// TIA Portal project "DP_Macko_2024" (V16)

(* hardware
DEVICE "S7-1200 station_1"  S7-1200 Station
   slot 0: "Rack_0"  S7-1200 Rack  Rack  V1.0
   slot 1: "PLC_1"  CPU 1214C DC/DC/DC  6ES7 214-1AG40-0XB0  V4.4
   slot 2: "DQ 16x24VDC_1"  SM 1222 DQ16 x 24VDC  6ES7 222-1BH32-0XB0  V2.0
DEVICE "ET 200SP station_1"  ET 200SP-Station
   slot 0: "Rack_0"  Rack  6ES5 710-8MAx1
   slot 0: "IO device_1"  IM 155-6 PN BA  6ES7 155-6AR00-0AN0  V3.2
   slot 1: "DI 16x24VDC ST_1"  DI 16x24VDC ST  6ES7 131-6BH00-0BA0  V1.1
      slot 1: "DI 16x24VDC ST_1"  DI 16x24VDC ST
   slot 2: "DI 16x24VDC ST_2"  DI 16x24VDC ST  6ES7 131-6BH00-0BA0  V1.1
      slot 1: "DI 16x24VDC ST_2"  DI 16x24VDC ST
   slot 3: "DQ 16x24VDC/0.5A BA_1"  DQ 16x24VDC/0.5A BA  6ES7 132-6BH00-0AA0  V0.0
      slot 1: "DQ 16x24VDC/0.5A BA_1"  DQ 16x24VDC/0.5A BA
   slot 4: "DQ 16x24VDC/0.5A BA_2"  DQ 16x24VDC/0.5A BA  6ES7 132-6BH00-0AA0  V0.0
      slot 1: "DQ 16x24VDC/0.5A BA_2"  DQ 16x24VDC/0.5A BA
   slot 5: "DQ 16x24VDC/0.5A BA_3"  DQ 16x24VDC/0.5A BA  6ES7 132-6BH00-0AA0  V0.0
      slot 1: "DQ 16x24VDC/0.5A BA_3"  DQ 16x24VDC/0.5A BA
   slot 6: "DQ 16x24VDC/0.5A BA_4"  DQ 16x24VDC/0.5A BA  6ES7 132-6BH00-0AA0  V0.0
      slot 1: "DQ 16x24VDC/0.5A BA_4"  DQ 16x24VDC/0.5A BA
   slot 7: "DQ 16x24VDC/0.5A BA_5"  DQ 16x24VDC/0.5A BA  6ES7 132-6BH00-0AA0  V0.0
      slot 1: "DQ 16x24VDC/0.5A BA_5"  DQ 16x24VDC/0.5A BA
   slot 8: "DQ 16x24VDC/0.5A BA_6"  DQ 16x24VDC/0.5A BA  6ES7 132-6BH00-0AA0  V0.0
      slot 1: "DQ 16x24VDC/0.5A BA_6"  DQ 16x24VDC/0.5A BA
   slot 9: "DQ 16x24VDC/0.5A BA_7"  DQ 16x24VDC/0.5A BA  6ES7 132-6BH00-0AA0  V0.0
      slot 1: "DQ 16x24VDC/0.5A BA_7"  DQ 16x24VDC/0.5A BA
   slot 10: "DQ 16x24VDC/0.5A BA_8"  DQ 16x24VDC/0.5A BA  6ES7 132-6BH00-0AA0  V0.0
      slot 1: "DQ 16x24VDC/0.5A BA_8"  DQ 16x24VDC/0.5A BA
   slot 11: "Server module_1"  Server module  6ES7 193-6PA00-0AA0  V1.1
      slot 1: "Server module_1"  Server module
   slot 127: "BA 2xRJ45"  BA 2xRJ45  6ES7 193-6AR00-0AA0  V0.0
      slot 1: "Port_1"  X1 P1 R  6ES7 193-6AR00-0AA0  V0.0
      slot 2: "Port_2"  X1 P2 R  6ES7 193-6AR00-0AA0  V0.0
DEVICE "S7300/ET200M station_1"  S7-300 station
   slot 0: "Rail_0"  Rail  6ES7 390-1***0-0AA0
   slot 2: "PLC_2"  CPU 313C-2 DP  6ES7 313-6CF03-0AB0  V2.6
      slot 0: "MPI interface_1"  X1
      slot 1: "DP interface_1"  X2
      slot 2: "DI 16/DO 16_1"  DI16/DO16
      slot 4: "Count_1"  Counter
   slot 4: "DI 16/DO 16x24VDC/0.5A_1"  DI16/DO16 x 24V / 0.5A  6ES7 323-1BL00-0AA0
   slot 5: "DO 16x24VDC/0.5A_1"  DO16 x 24VDC / 0.5A  6ES7 322-1BH01-0AA0
*)

// ===== PLC "PLC_2"  CPU 313C-2 DP =====

VAR_GLOBAL   // PLC tag table "kolajove_obvody"
   "3k1" AT %I124.4 : Bool;
   "3k2" AT %I124.5 : Bool;
   "4k1" AT %I124.6 : Bool;
   "4k2" AT %I124.7 : Bool;
   "5k1" AT %I125.0 : Bool;
   "5k2" AT %I125.1 : Bool;
   "9k2" AT %I0.1 : Bool;
   "10k1" AT %I0.2 : Bool;
   "10k2" AT %I0.3 : Bool;
   "11k1" AT %I0.4 : Bool;
   "11k2" AT %I0.5 : Bool;
   "8k2" AT %I125.7 : Bool;
   "9k1" AT %I0.0 : Bool;
   "12k1" AT %I0.6 : Bool;
   "12k2" AT %I0.7 : Bool;
   "2k1" AT %I124.2 : Bool;
   "2k2" AT %I124.3 : Bool;
   "6k1" AT %I125.2 : Bool;
   "6k2" AT %I125.3 : Bool;
   "7k1" AT %I125.4 : Bool;
   "14k1" AT %I1.2 : Bool;
   "1k1" AT %I124.0 : Bool;
   "1k2" AT %I124.1 : Bool;
   "7k2" AT %I125.5 : Bool;
   "8k1" AT %I125.6 : Bool;
   "13k1" AT %I1.0 : Bool;
   "13k2" AT %I1.1 : Bool;
   "14k2" AT %I1.3 : Bool;
   "RAD_k1" AT %Q124.0 : Bool;
   "RAD_k2" AT %Q124.1 : Bool;
   "RAD_v1" AT %Q124.2 : Bool;
   "RAD_Sk" AT %Q124.3 : Bool;
   "TU_RAD_ZBE_1" AT %Q124.4 : Bool;
   "TU_RAD_ZBE_2" AT %Q124.5 : Bool;
   "TU_RAD_ZBE_3" AT %Q124.6 : Bool;
   "TU_RAD_ZBE_4" AT %Q124.7 : Bool;
   "ZBE_Lk" AT %Q125.0 : Bool;
   "ZBE_BLk" AT %Q125.1 : Bool;
   "ZBE_v1" AT %Q125.2 : Bool;
   "ZBE_v2" AT %Q125.3 : Bool;
   "ZBE_k1" AT %Q125.4 : Bool;
   "ZBE_k2" AT %Q125.5 : Bool;
   "ZBE_v3" AT %Q125.6 : Bool;
   "ZBE_Sk" AT %Q125.7 : Bool;
   "TU_ZBE_HLO_1" AT %Q0.0 : Bool;
   "TU_ZBE_HLO_2" AT %Q0.1 : Bool;
   "HLO_Lk" AT %Q0.2 : Bool;
   "HLO_v1" AT %Q0.3 : Bool;
   "HLO_k1" AT %Q0.4 : Bool;
   "HLO_k2" AT %Q0.5 : Bool;
   "C_PU1" AT %Q0.7 : Bool;
   "C_AU" AT %Q1.0 : Bool;
   "C_PU2" AT %Q1.1 : Bool;
   "E_PU1" AT %Q1.2 : Bool;
   "E_AU" AT %Q1.3 : Bool;
   "E_PU2" AT %Q1.4 : Bool;
   "OD_ZBE_HLO" AT %Q1.5 : Bool;
END_VAR

DATA_BLOCK "Tratove_useky_DB"   // DB1
{ S7_Optimized_Access := 'FALSE' }
VERSION : 0.1
// stored: InstanceOfName Tratove_useky
"Tratove_useky"
BEGIN
END_DATA_BLOCK

FUNCTION_BLOCK "Tratove_useky"   // FB1, LAD
{ S7_Optimized_Access := 'FALSE' }
VERSION : 0.1
   VAR_INPUT
      RAD_1 : Bool;
      RAD_2 : Bool;
      RAD_3 : Bool;
      RAD_4 : Bool;
      RAD_5 : Bool;
      RAD_ZBE_1 : Bool;
      RAD_ZBE_2 : Bool;
      RAD_ZBE_3 : Bool;
      RAD_ZBE_4 : Bool;
      RAD_ZBE_5 : Bool;
      ZBE_1 : Bool;
      ZBE_2 : Bool;
      ZBE_3 : Bool;
      ZBE_4 : Bool;
      ZBE_5 : Bool;
      ZBE_6 : Bool;
      ZBE_7 : Bool;
      ZBE_8 : Bool;
      ZBE_HLO_1 : Bool;
      ZBE_HLO_2 : Bool;
      ZBE_HLO_3 : Bool;
      ZBE_HLO_4 : Bool;
      ZBE_HLO_5 : Bool;
      ZBE_HLO_6 : Bool;
      HLO_1 : Bool;
      HLO_2 : Bool;
      HLO_3 : Bool;
      HLO_4 : Bool;
   END_VAR
   VAR_OUTPUT
      RAD_k1 : Bool;
      RAD_k2 : Bool;
      RAD_v1 : Bool;
      RAD_Sk : Bool;
      TU_RAD_ZBE_1 : Bool;
      TU_RAD_ZBE_2 : Bool;
      TU_RAD_ZBE_3 : Bool;
      TU_RAD_ZBE_4 : Bool;
      ZBE_Lk : Bool;
      ZBE_BLk : Bool;
      ZBE_v1 : Bool;
      ZBE_v2 : Bool;
      ZBE_k1 : Bool;
      ZBE_k2 : Bool;
      ZBE_v3 : Bool;
      ZBE_Sk : Bool;
      TU_ZBE_HLO_1 : Bool;
      OD_ZBE_HLO : Bool;
      TU_ZBE_HLO_2 : Bool;
      HLO_Lk : Bool;
      HLO_v1 : Bool;
      HLO_k1 : Bool;
      HLO_k2 : Bool;
      C_PU1 : Bool;
      C_AU : Bool;
      C_PU2 : Bool;
      E_PU1 : Bool;
      E_AU : Bool;
      E_PU2 : Bool;
   END_VAR
   VAR
      cRAD_k1 : TON;
      cRAD_k2 : TON;
      cRAD_v1 : TON;
      cRAD_Sk : TON;
      cTU_RAD_ZBE_1 : TON;
      cTU_RAD_ZBE_2 : TON;
      cTU_RAD_ZBE_3 : TON;
      cTU_RAD_ZBE_4 : TON;
      cZBE_Lk : TON;
      cZBE_BLk : TON;
      cZBE_v1 : TON;
      cZBE_v2 : TON;
      cZBE_k1 : TON;
      cZBE_k2 : TON;
      cZBE_v3 : TON;
      cZBE_Sk : TON;
      cTU_ZBE_HLO_1 : TON;
      cOD_ZBE_HLO : TON;
      cTU_ZBE_HLO_2 : TON;
      cHLO_k1 : TON;
      cHLO_k2 : TON;
      cHLO_v1 : TON;
      cHLO_Lk : TON;
      cC_PU1 : TON;
      cC_AU : TON;
      cC_PU2 : TON;
      cE_PU1 : TON;
      cE_AU : TON;
      cE_PU2 : TON;
      oneskorenie : Time := T#250ms;
      cRAD_k1_Off : TON;
      cRAD_k2_Off : TON;
      cRAD_v1_Off : TON;
      cRAD_Sk_Off : TON;
      cTU_RAD_ZBE_1_Off : TON;
      cTU_RAD_ZBE_2_Off : TON;
      cTU_RAD_ZBE_3_Off : TON;
      cTU_RAD_ZBE_4_Off : TON;
      cZBE_Lk_Off : TON;
      cZBE_BLk_Off : TON;
      cZBE_v1_Off : TON;
      cZBE_v2_Off : TON;
      cZBE_k1_Off : TON;
      cZBE_k2_Off : TON;
      cZBE_v3_Off : TON;
      cZBE_Sk_Off : TON;
      cTU_ZBE_HLO_1_Off : TON;
      cOD_ZBE_HLO_Off : TON;
      cTU_ZBE_HLO_2_Off : TON;
      cHLO_k1_Off : TON;
      cHLO_k2_Off : TON;
      cHLO_v1_Off : TON;
      cHLO_Lk_Off : TON;
      cC_PU1_Off : TON;
      cC_AU_Off : TON;
      cC_PU2_Off : TON;
      cE_PU1_Off : TON;
      cE_AU_Off : TON;
      cE_PU2_Off : TON;
   END_VAR
BEGIN

REGION Network 1: Casovac RAD_k1
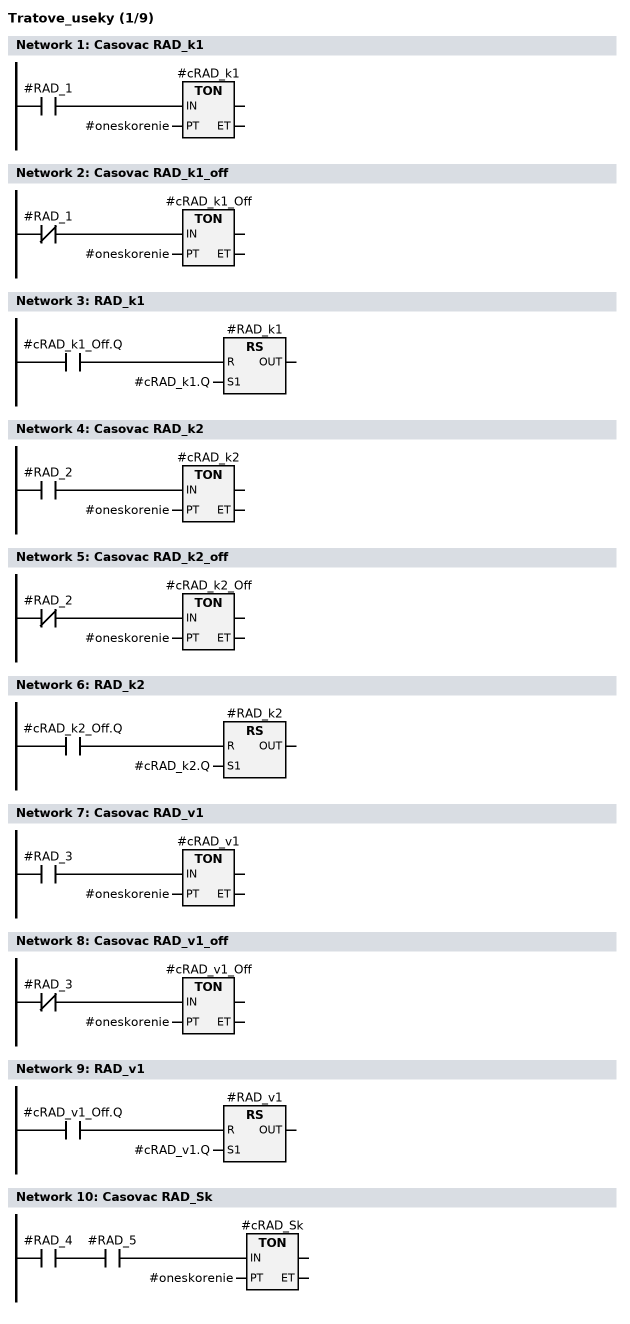
   #cRAD_k1.TON(IN := #RAD_1, PT := #oneskorenie);
END_REGION

REGION Network 2: Casovac RAD_k1_off
   #cRAD_k1_Off.TON(IN := NOT #RAD_1, PT := #oneskorenie);
END_REGION

REGION Network 3: RAD_k1
   RUNG wire#powerrail
      Contact( #cRAD_k1_Off.Q )
      S_RS(operand := #RAD_k1, s1 := #cRAD_k1.Q)
   END_RUNG
   // the same network as SCL:
   IF #cRAD_k1_Off.Q THEN
       #RAD_k1 := FALSE;   // RS flip-flop
   END_IF;
   IF #cRAD_k1.Q THEN #RAD_k1 := TRUE; END_IF;
END_REGION

REGION Network 4: Casovac RAD_k2
   #cRAD_k2.TON(IN := #RAD_2, PT := #oneskorenie);
END_REGION

REGION Network 5: Casovac RAD_k2_off
   #cRAD_k2_Off.TON(IN := NOT #RAD_2, PT := #oneskorenie);
END_REGION

REGION Network 6: RAD_k2
   RUNG wire#powerrail
      Contact( #cRAD_k2_Off.Q )
      S_RS(operand := #RAD_k2, s1 := #cRAD_k2.Q)
   END_RUNG
   // the same network as SCL:
   IF #cRAD_k2_Off.Q THEN
       #RAD_k2 := FALSE;   // RS flip-flop
   END_IF;
   IF #cRAD_k2.Q THEN #RAD_k2 := TRUE; END_IF;
END_REGION

REGION Network 7: Casovac RAD_v1
   #cRAD_v1.TON(IN := #RAD_3, PT := #oneskorenie);
END_REGION

REGION Network 8: Casovac RAD_v1_off
   #cRAD_v1_Off.TON(IN := NOT #RAD_3, PT := #oneskorenie);
END_REGION

REGION Network 9: RAD_v1
   RUNG wire#powerrail
      Contact( #cRAD_v1_Off.Q )
      S_RS(operand := #RAD_v1, s1 := #cRAD_v1.Q)
   END_RUNG
   // the same network as SCL:
   IF #cRAD_v1_Off.Q THEN
       #RAD_v1 := FALSE;   // RS flip-flop
   END_IF;
   IF #cRAD_v1.Q THEN #RAD_v1 := TRUE; END_IF;
END_REGION

REGION Network 10: Casovac RAD_Sk
   #cRAD_Sk.TON(IN := #RAD_4 AND #RAD_5, PT := #oneskorenie);
END_REGION

REGION Network 11: Casovac RAD_Sk_off
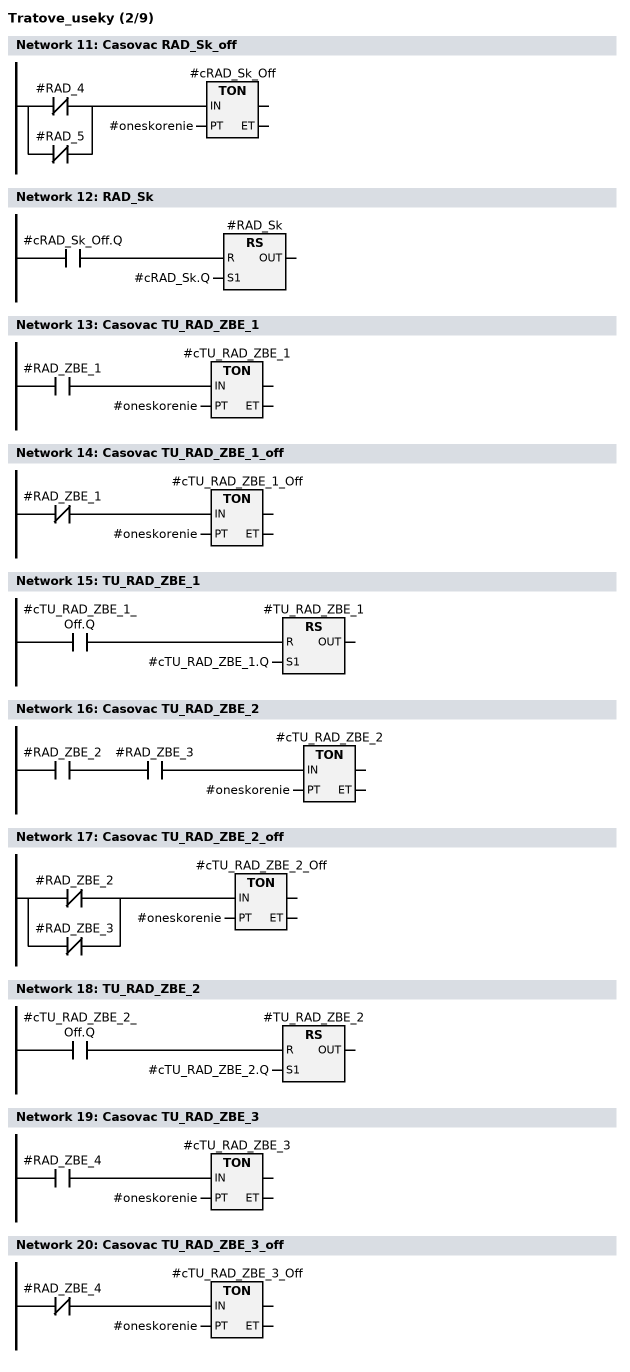
   #cRAD_Sk_Off.TON(IN := NOT #RAD_4 OR NOT #RAD_5, PT := #oneskorenie);
END_REGION

REGION Network 12: RAD_Sk
   RUNG wire#powerrail
      Contact( #cRAD_Sk_Off.Q )
      S_RS(operand := #RAD_Sk, s1 := #cRAD_Sk.Q)
   END_RUNG
   // the same network as SCL:
   IF #cRAD_Sk_Off.Q THEN
       #RAD_Sk := FALSE;   // RS flip-flop
   END_IF;
   IF #cRAD_Sk.Q THEN #RAD_Sk := TRUE; END_IF;
END_REGION

REGION Network 13: Casovac TU_RAD_ZBE_1
   #cTU_RAD_ZBE_1.TON(IN := #RAD_ZBE_1, PT := #oneskorenie);
END_REGION

REGION Network 14: Casovac TU_RAD_ZBE_1_off
   #cTU_RAD_ZBE_1_Off.TON(IN := NOT #RAD_ZBE_1, PT := #oneskorenie);
END_REGION

REGION Network 15: TU_RAD_ZBE_1
   RUNG wire#powerrail
      Contact( #cTU_RAD_ZBE_1_Off.Q )
      S_RS(operand := #TU_RAD_ZBE_1, s1 := #cTU_RAD_ZBE_1.Q)
   END_RUNG
   // the same network as SCL:
   IF #cTU_RAD_ZBE_1_Off.Q THEN
       #TU_RAD_ZBE_1 := FALSE;   // RS flip-flop
   END_IF;
   IF #cTU_RAD_ZBE_1.Q THEN #TU_RAD_ZBE_1 := TRUE; END_IF;
END_REGION

REGION Network 16: Casovac TU_RAD_ZBE_2
   #cTU_RAD_ZBE_2.TON(IN := #RAD_ZBE_2 AND #RAD_ZBE_3, PT := #oneskorenie);
END_REGION

REGION Network 17: Casovac TU_RAD_ZBE_2_off
   #cTU_RAD_ZBE_2_Off.TON(IN := NOT #RAD_ZBE_2 OR NOT #RAD_ZBE_3, PT := #oneskorenie);
END_REGION

REGION Network 18: TU_RAD_ZBE_2
   RUNG wire#powerrail
      Contact( #cTU_RAD_ZBE_2_Off.Q )
      S_RS(operand := #TU_RAD_ZBE_2, s1 := #cTU_RAD_ZBE_2.Q)
   END_RUNG
   // the same network as SCL:
   IF #cTU_RAD_ZBE_2_Off.Q THEN
       #TU_RAD_ZBE_2 := FALSE;   // RS flip-flop
   END_IF;
   IF #cTU_RAD_ZBE_2.Q THEN #TU_RAD_ZBE_2 := TRUE; END_IF;
END_REGION

REGION Network 19: Casovac TU_RAD_ZBE_3
   #cTU_RAD_ZBE_3.TON(IN := #RAD_ZBE_4, PT := #oneskorenie);
END_REGION

REGION Network 20: Casovac TU_RAD_ZBE_3_off
   #cTU_RAD_ZBE_3_Off.TON(IN := NOT #RAD_ZBE_4, PT := #oneskorenie);
END_REGION

REGION Network 21: TU_RAD_ZBE_3
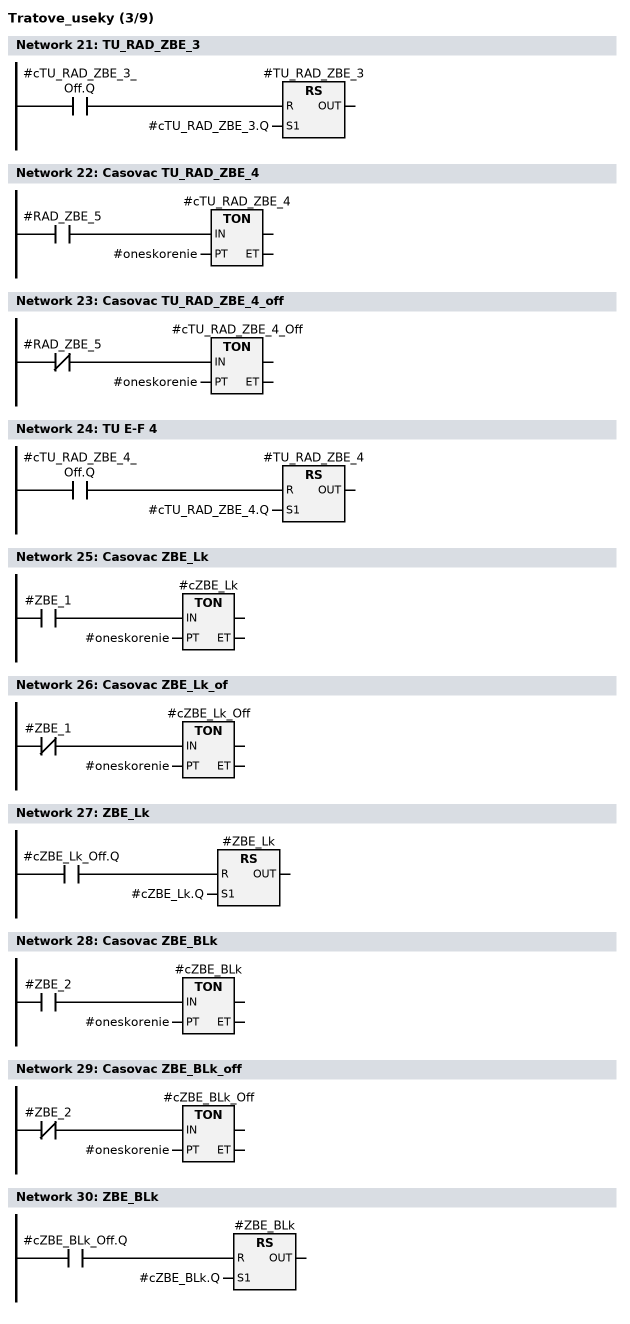
   RUNG wire#powerrail
      Contact( #cTU_RAD_ZBE_3_Off.Q )
      S_RS(operand := #TU_RAD_ZBE_3, s1 := #cTU_RAD_ZBE_3.Q)
   END_RUNG
   // the same network as SCL:
   IF #cTU_RAD_ZBE_3_Off.Q THEN
       #TU_RAD_ZBE_3 := FALSE;   // RS flip-flop
   END_IF;
   IF #cTU_RAD_ZBE_3.Q THEN #TU_RAD_ZBE_3 := TRUE; END_IF;
END_REGION

REGION Network 22: Casovac TU_RAD_ZBE_4
   #cTU_RAD_ZBE_4.TON(IN := #RAD_ZBE_5, PT := #oneskorenie);
END_REGION

REGION Network 23: Casovac TU_RAD_ZBE_4_off
   #cTU_RAD_ZBE_4_Off.TON(IN := NOT #RAD_ZBE_5, PT := #oneskorenie);
END_REGION

REGION Network 24: TU E-F 4
   RUNG wire#powerrail
      Contact( #cTU_RAD_ZBE_4_Off.Q )
      S_RS(operand := #TU_RAD_ZBE_4, s1 := #cTU_RAD_ZBE_4.Q)
   END_RUNG
   // the same network as SCL:
   IF #cTU_RAD_ZBE_4_Off.Q THEN
       #TU_RAD_ZBE_4 := FALSE;   // RS flip-flop
   END_IF;
   IF #cTU_RAD_ZBE_4.Q THEN #TU_RAD_ZBE_4 := TRUE; END_IF;
END_REGION

REGION Network 25: Casovac ZBE_Lk
   #cZBE_Lk.TON(IN := #ZBE_1, PT := #oneskorenie);
END_REGION

REGION Network 26: Casovac ZBE_Lk_of
   #cZBE_Lk_Off.TON(IN := NOT #ZBE_1, PT := #oneskorenie);
END_REGION

REGION Network 27: ZBE_Lk
   RUNG wire#powerrail
      Contact( #cZBE_Lk_Off.Q )
      S_RS(operand := #ZBE_Lk, s1 := #cZBE_Lk.Q)
   END_RUNG
   // the same network as SCL:
   IF #cZBE_Lk_Off.Q THEN
       #ZBE_Lk := FALSE;   // RS flip-flop
   END_IF;
   IF #cZBE_Lk.Q THEN #ZBE_Lk := TRUE; END_IF;
END_REGION

REGION Network 28: Casovac ZBE_BLk
   #cZBE_BLk.TON(IN := #ZBE_2, PT := #oneskorenie);
END_REGION

REGION Network 29: Casovac ZBE_BLk_off
   #cZBE_BLk_Off.TON(IN := NOT #ZBE_2, PT := #oneskorenie);
END_REGION

REGION Network 30: ZBE_BLk
   RUNG wire#powerrail
      Contact( #cZBE_BLk_Off.Q )
      S_RS(operand := #ZBE_BLk, s1 := #cZBE_BLk.Q)
   END_RUNG
   // the same network as SCL:
   IF #cZBE_BLk_Off.Q THEN
       #ZBE_BLk := FALSE;   // RS flip-flop
   END_IF;
   IF #cZBE_BLk.Q THEN #ZBE_BLk := TRUE; END_IF;
END_REGION

REGION Network 31: Casovac ZBE_v1
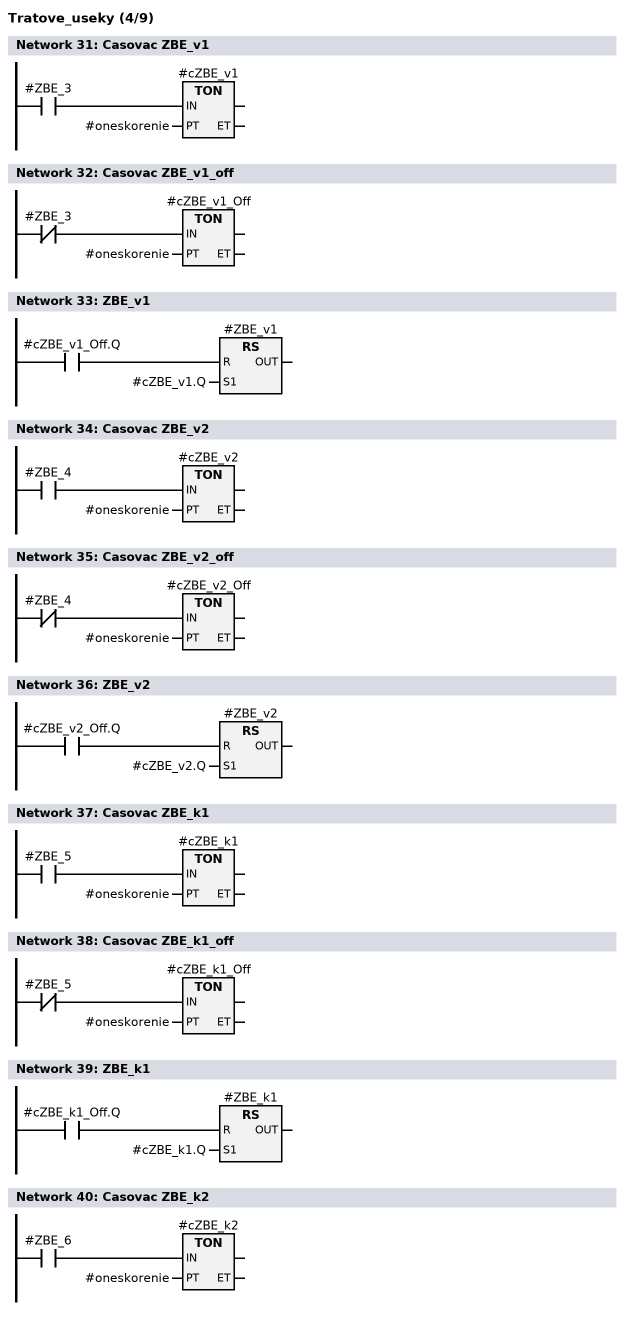
   #cZBE_v1.TON(IN := #ZBE_3, PT := #oneskorenie);
END_REGION

REGION Network 32: Casovac ZBE_v1_off
   #cZBE_v1_Off.TON(IN := NOT #ZBE_3, PT := #oneskorenie);
END_REGION

REGION Network 33: ZBE_v1
   RUNG wire#powerrail
      Contact( #cZBE_v1_Off.Q )
      S_RS(operand := #ZBE_v1, s1 := #cZBE_v1.Q)
   END_RUNG
   // the same network as SCL:
   IF #cZBE_v1_Off.Q THEN
       #ZBE_v1 := FALSE;   // RS flip-flop
   END_IF;
   IF #cZBE_v1.Q THEN #ZBE_v1 := TRUE; END_IF;
END_REGION

REGION Network 34: Casovac ZBE_v2
   #cZBE_v2.TON(IN := #ZBE_4, PT := #oneskorenie);
END_REGION

REGION Network 35: Casovac ZBE_v2_off
   #cZBE_v2_Off.TON(IN := NOT #ZBE_4, PT := #oneskorenie);
END_REGION

REGION Network 36: ZBE_v2
   RUNG wire#powerrail
      Contact( #cZBE_v2_Off.Q )
      S_RS(operand := #ZBE_v2, s1 := #cZBE_v2.Q)
   END_RUNG
   // the same network as SCL:
   IF #cZBE_v2_Off.Q THEN
       #ZBE_v2 := FALSE;   // RS flip-flop
   END_IF;
   IF #cZBE_v2.Q THEN #ZBE_v2 := TRUE; END_IF;
END_REGION

REGION Network 37: Casovac ZBE_k1
   #cZBE_k1.TON(IN := #ZBE_5, PT := #oneskorenie);
END_REGION

REGION Network 38: Casovac ZBE_k1_off
   #cZBE_k1_Off.TON(IN := NOT #ZBE_5, PT := #oneskorenie);
END_REGION

REGION Network 39: ZBE_k1
   RUNG wire#powerrail
      Contact( #cZBE_k1_Off.Q )
      S_RS(operand := #ZBE_k1, s1 := #cZBE_k1.Q)
   END_RUNG
   // the same network as SCL:
   IF #cZBE_k1_Off.Q THEN
       #ZBE_k1 := FALSE;   // RS flip-flop
   END_IF;
   IF #cZBE_k1.Q THEN #ZBE_k1 := TRUE; END_IF;
END_REGION

REGION Network 40: Casovac ZBE_k2
   #cZBE_k2.TON(IN := #ZBE_6, PT := #oneskorenie);
END_REGION

REGION Network 41: Casovac ZBE_k2_off
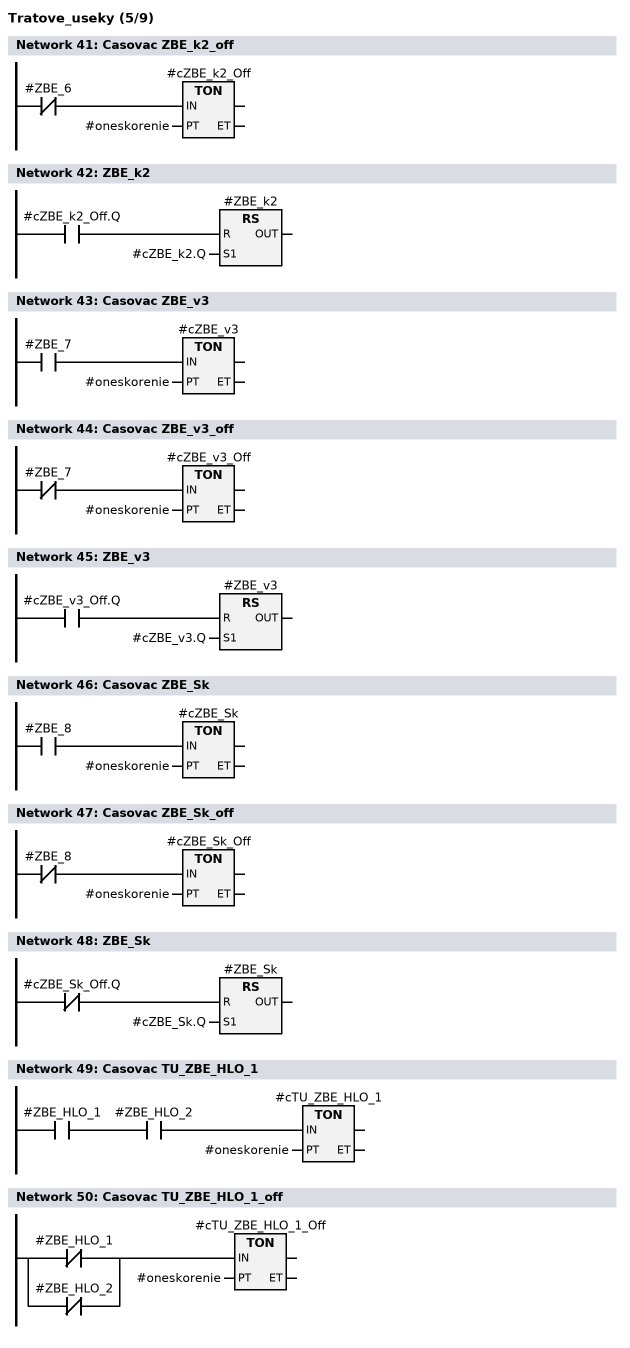
   #cZBE_k2_Off.TON(IN := NOT #ZBE_6, PT := #oneskorenie);
END_REGION

REGION Network 42: ZBE_k2
   RUNG wire#powerrail
      Contact( #cZBE_k2_Off.Q )
      S_RS(operand := #ZBE_k2, s1 := #cZBE_k2.Q)
   END_RUNG
   // the same network as SCL:
   IF #cZBE_k2_Off.Q THEN
       #ZBE_k2 := FALSE;   // RS flip-flop
   END_IF;
   IF #cZBE_k2.Q THEN #ZBE_k2 := TRUE; END_IF;
END_REGION

REGION Network 43: Casovac ZBE_v3
   #cZBE_v3.TON(IN := #ZBE_7, PT := #oneskorenie);
END_REGION

REGION Network 44: Casovac ZBE_v3_off
   #cZBE_v3_Off.TON(IN := NOT #ZBE_7, PT := #oneskorenie);
END_REGION

REGION Network 45: ZBE_v3
   RUNG wire#powerrail
      Contact( #cZBE_v3_Off.Q )
      S_RS(operand := #ZBE_v3, s1 := #cZBE_v3.Q)
   END_RUNG
   // the same network as SCL:
   IF #cZBE_v3_Off.Q THEN
       #ZBE_v3 := FALSE;   // RS flip-flop
   END_IF;
   IF #cZBE_v3.Q THEN #ZBE_v3 := TRUE; END_IF;
END_REGION

REGION Network 46: Casovac ZBE_Sk
   #cZBE_Sk.TON(IN := #ZBE_8, PT := #oneskorenie);
END_REGION

REGION Network 47: Casovac ZBE_Sk_off
   #cZBE_Sk_Off.TON(IN := NOT #ZBE_8, PT := #oneskorenie);
END_REGION

REGION Network 48: ZBE_Sk
   RUNG wire#powerrail
      I_Contact( #cZBE_Sk_Off.Q )
      S_RS(operand := #ZBE_Sk, s1 := #cZBE_Sk.Q)
   END_RUNG
   // the same network as SCL:
   IF NOT #cZBE_Sk_Off.Q THEN
       #ZBE_Sk := FALSE;   // RS flip-flop
   END_IF;
   IF #cZBE_Sk.Q THEN #ZBE_Sk := TRUE; END_IF;
END_REGION

REGION Network 49: Casovac TU_ZBE_HLO_1
   #cTU_ZBE_HLO_1.TON(IN := #ZBE_HLO_1 AND #ZBE_HLO_2, PT := #oneskorenie);
END_REGION

REGION Network 50: Casovac TU_ZBE_HLO_1_off
   #cTU_ZBE_HLO_1_Off.TON(IN := NOT #ZBE_HLO_1 OR NOT #ZBE_HLO_2, PT := #oneskorenie);
END_REGION

REGION Network 51: TU_ZBE_HLO_1
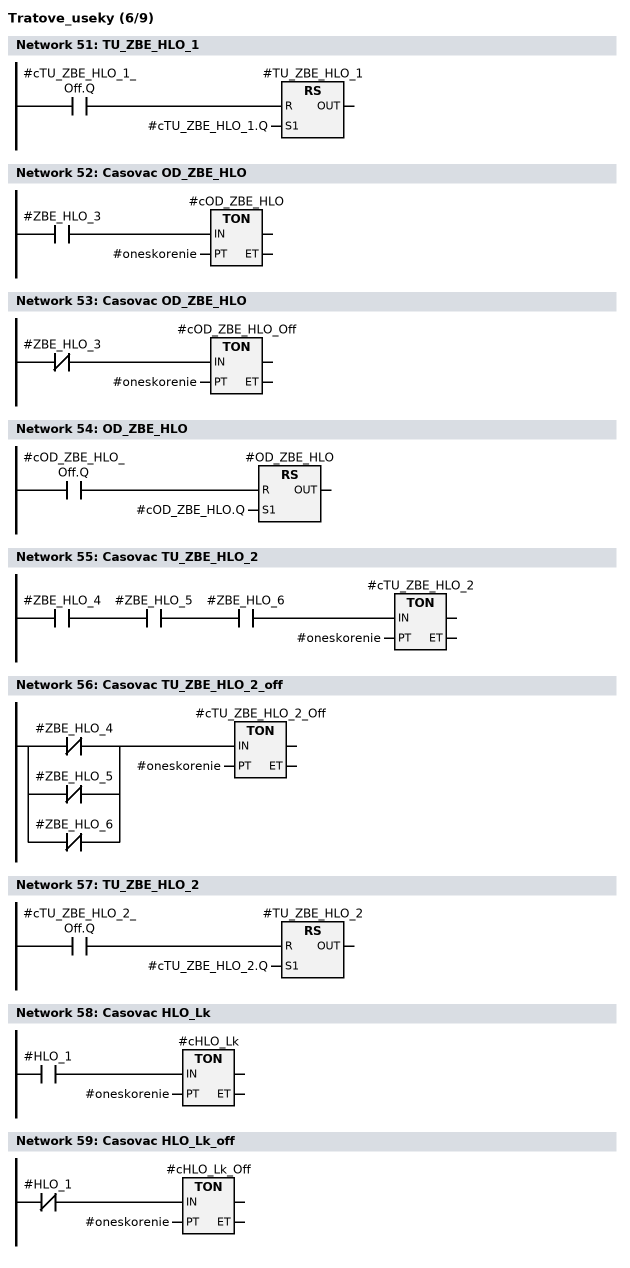
   RUNG wire#powerrail
      Contact( #cTU_ZBE_HLO_1_Off.Q )
      S_RS(operand := #TU_ZBE_HLO_1, s1 := #cTU_ZBE_HLO_1.Q)
   END_RUNG
   // the same network as SCL:
   IF #cTU_ZBE_HLO_1_Off.Q THEN
       #TU_ZBE_HLO_1 := FALSE;   // RS flip-flop
   END_IF;
   IF #cTU_ZBE_HLO_1.Q THEN #TU_ZBE_HLO_1 := TRUE; END_IF;
END_REGION

REGION Network 52: Casovac OD_ZBE_HLO
   #cOD_ZBE_HLO.TON(IN := #ZBE_HLO_3, PT := #oneskorenie);
END_REGION

REGION Network 53: Casovac OD_ZBE_HLO
   #cOD_ZBE_HLO_Off.TON(IN := NOT #ZBE_HLO_3, PT := #oneskorenie);
END_REGION

REGION Network 54: OD_ZBE_HLO
   RUNG wire#powerrail
      Contact( #cOD_ZBE_HLO_Off.Q )
      S_RS(operand := #OD_ZBE_HLO, s1 := #cOD_ZBE_HLO.Q)
   END_RUNG
   // the same network as SCL:
   IF #cOD_ZBE_HLO_Off.Q THEN
       #OD_ZBE_HLO := FALSE;   // RS flip-flop
   END_IF;
   IF #cOD_ZBE_HLO.Q THEN #OD_ZBE_HLO := TRUE; END_IF;
END_REGION

REGION Network 55: Casovac TU_ZBE_HLO_2
   #cTU_ZBE_HLO_2.TON(IN := #ZBE_HLO_4 AND #ZBE_HLO_5 AND #ZBE_HLO_6, PT := #oneskorenie);
END_REGION

REGION Network 56: Casovac TU_ZBE_HLO_2_off
   #cTU_ZBE_HLO_2_Off.TON(IN := NOT #ZBE_HLO_4 OR NOT #ZBE_HLO_5 OR NOT #ZBE_HLO_6, PT := #oneskorenie);
END_REGION

REGION Network 57: TU_ZBE_HLO_2
   RUNG wire#powerrail
      Contact( #cTU_ZBE_HLO_2_Off.Q )
      S_RS(operand := #TU_ZBE_HLO_2, s1 := #cTU_ZBE_HLO_2.Q)
   END_RUNG
   // the same network as SCL:
   IF #cTU_ZBE_HLO_2_Off.Q THEN
       #TU_ZBE_HLO_2 := FALSE;   // RS flip-flop
   END_IF;
   IF #cTU_ZBE_HLO_2.Q THEN #TU_ZBE_HLO_2 := TRUE; END_IF;
END_REGION

REGION Network 58: Casovac HLO_Lk
   #cHLO_Lk.TON(IN := #HLO_1, PT := #oneskorenie);
END_REGION

REGION Network 59: Casovac HLO_Lk_off
   #cHLO_Lk_Off.TON(IN := NOT #HLO_1, PT := #oneskorenie);
END_REGION

REGION Network 60: HLO_Lk
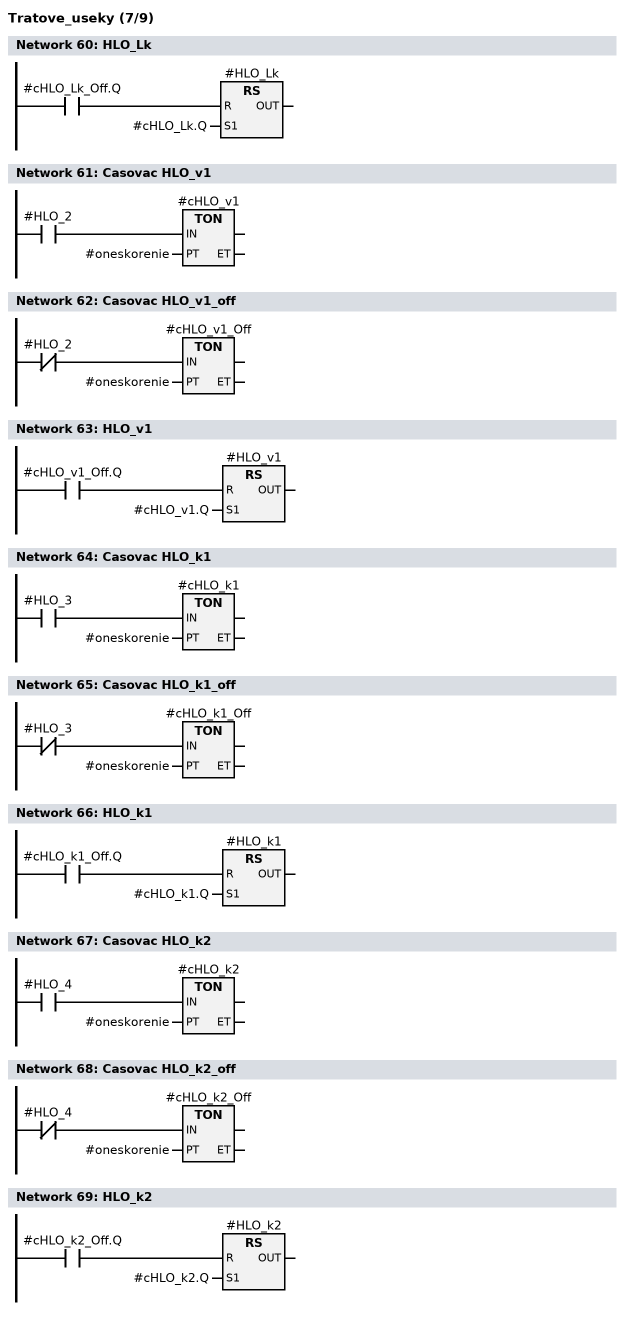
   RUNG wire#powerrail
      Contact( #cHLO_Lk_Off.Q )
      S_RS(operand := #HLO_Lk, s1 := #cHLO_Lk.Q)
   END_RUNG
   // the same network as SCL:
   IF #cHLO_Lk_Off.Q THEN
       #HLO_Lk := FALSE;   // RS flip-flop
   END_IF;
   IF #cHLO_Lk.Q THEN #HLO_Lk := TRUE; END_IF;
END_REGION

REGION Network 61: Casovac HLO_v1
   #cHLO_v1.TON(IN := #HLO_2, PT := #oneskorenie);
END_REGION

REGION Network 62: Casovac HLO_v1_off
   #cHLO_v1_Off.TON(IN := NOT #HLO_2, PT := #oneskorenie);
END_REGION

REGION Network 63: HLO_v1
   RUNG wire#powerrail
      Contact( #cHLO_v1_Off.Q )
      S_RS(operand := #HLO_v1, s1 := #cHLO_v1.Q)
   END_RUNG
   // the same network as SCL:
   IF #cHLO_v1_Off.Q THEN
       #HLO_v1 := FALSE;   // RS flip-flop
   END_IF;
   IF #cHLO_v1.Q THEN #HLO_v1 := TRUE; END_IF;
END_REGION

REGION Network 64: Casovac HLO_k1
   #cHLO_k1.TON(IN := #HLO_3, PT := #oneskorenie);
END_REGION

REGION Network 65: Casovac HLO_k1_off
   #cHLO_k1_Off.TON(IN := NOT #HLO_3, PT := #oneskorenie);
END_REGION

REGION Network 66: HLO_k1
   RUNG wire#powerrail
      Contact( #cHLO_k1_Off.Q )
      S_RS(operand := #HLO_k1, s1 := #cHLO_k1.Q)
   END_RUNG
   // the same network as SCL:
   IF #cHLO_k1_Off.Q THEN
       #HLO_k1 := FALSE;   // RS flip-flop
   END_IF;
   IF #cHLO_k1.Q THEN #HLO_k1 := TRUE; END_IF;
END_REGION

REGION Network 67: Casovac HLO_k2
   #cHLO_k2.TON(IN := #HLO_4, PT := #oneskorenie);
END_REGION

REGION Network 68: Casovac HLO_k2_off
   #cHLO_k2_Off.TON(IN := NOT #HLO_4, PT := #oneskorenie);
END_REGION

REGION Network 69: HLO_k2
   RUNG wire#powerrail
      Contact( #cHLO_k2_Off.Q )
      S_RS(operand := #HLO_k2, s1 := #cHLO_k2.Q)
   END_RUNG
   // the same network as SCL:
   IF #cHLO_k2_Off.Q THEN
       #HLO_k2 := FALSE;   // RS flip-flop
   END_IF;
   IF #cHLO_k2.Q THEN #HLO_k2 := TRUE; END_IF;
END_REGION

REGION Network 70: Casovac C_PU1
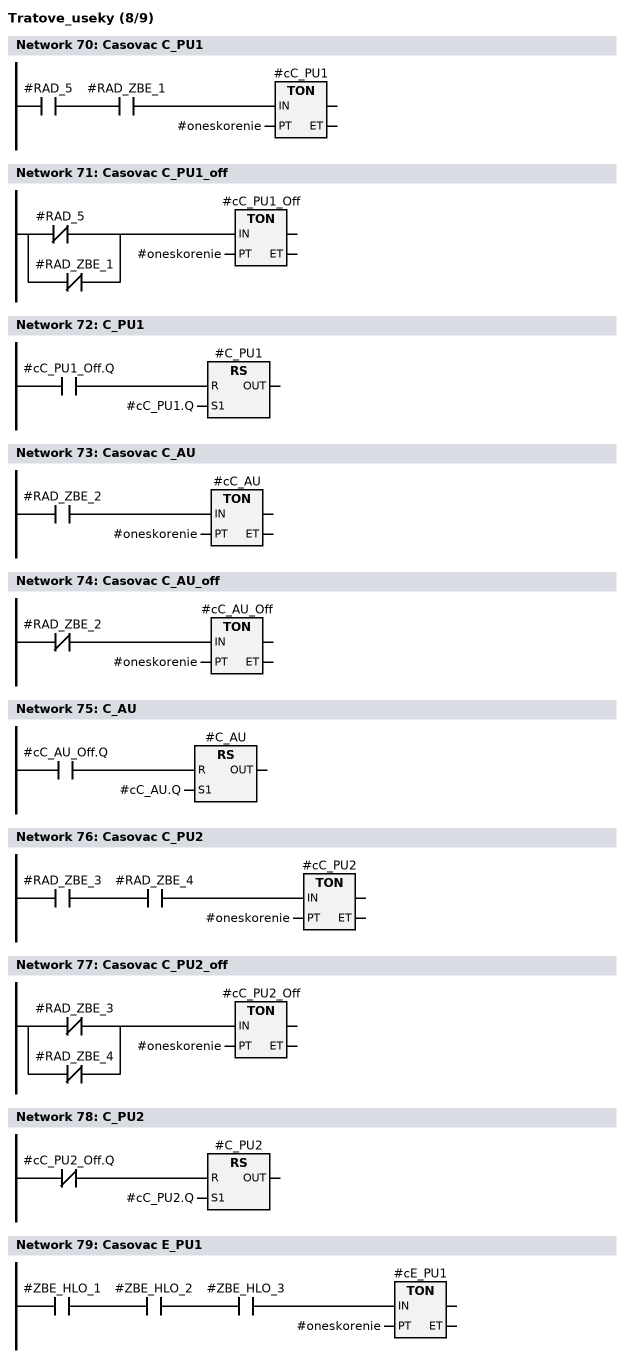
   #cC_PU1.TON(IN := #RAD_5 AND #RAD_ZBE_1, PT := #oneskorenie);
END_REGION

REGION Network 71: Casovac C_PU1_off
   #cC_PU1_Off.TON(IN := NOT #RAD_5 OR NOT #RAD_ZBE_1, PT := #oneskorenie);
END_REGION

REGION Network 72: C_PU1
   RUNG wire#powerrail
      Contact( #cC_PU1_Off.Q )
      S_RS(operand := #C_PU1, s1 := #cC_PU1.Q)
   END_RUNG
   // the same network as SCL:
   IF #cC_PU1_Off.Q THEN
       #C_PU1 := FALSE;   // RS flip-flop
   END_IF;
   IF #cC_PU1.Q THEN #C_PU1 := TRUE; END_IF;
END_REGION

REGION Network 73: Casovac C_AU
   #cC_AU.TON(IN := #RAD_ZBE_2, PT := #oneskorenie);
END_REGION

REGION Network 74: Casovac C_AU_off
   #cC_AU_Off.TON(IN := NOT #RAD_ZBE_2, PT := #oneskorenie);
END_REGION

REGION Network 75: C_AU
   RUNG wire#powerrail
      Contact( #cC_AU_Off.Q )
      S_RS(operand := #C_AU, s1 := #cC_AU.Q)
   END_RUNG
   // the same network as SCL:
   IF #cC_AU_Off.Q THEN
       #C_AU := FALSE;   // RS flip-flop
   END_IF;
   IF #cC_AU.Q THEN #C_AU := TRUE; END_IF;
END_REGION

REGION Network 76: Casovac C_PU2
   #cC_PU2.TON(IN := #RAD_ZBE_3 AND #RAD_ZBE_4, PT := #oneskorenie);
END_REGION

REGION Network 77: Casovac C_PU2_off
   #cC_PU2_Off.TON(IN := NOT #RAD_ZBE_3 OR NOT #RAD_ZBE_4, PT := #oneskorenie);
END_REGION

REGION Network 78: C_PU2
   RUNG wire#powerrail
      I_Contact( #cC_PU2_Off.Q )
      S_RS(operand := #C_PU2, s1 := #cC_PU2.Q)
   END_RUNG
   // the same network as SCL:
   IF NOT #cC_PU2_Off.Q THEN
       #C_PU2 := FALSE;   // RS flip-flop
   END_IF;
   IF #cC_PU2.Q THEN #C_PU2 := TRUE; END_IF;
END_REGION

REGION Network 79: Casovac E_PU1
   #cE_PU1.TON(IN := #ZBE_HLO_1 AND #ZBE_HLO_2 AND #ZBE_HLO_3, PT := #oneskorenie);
END_REGION

REGION Network 80: Casovac E_PU1_off
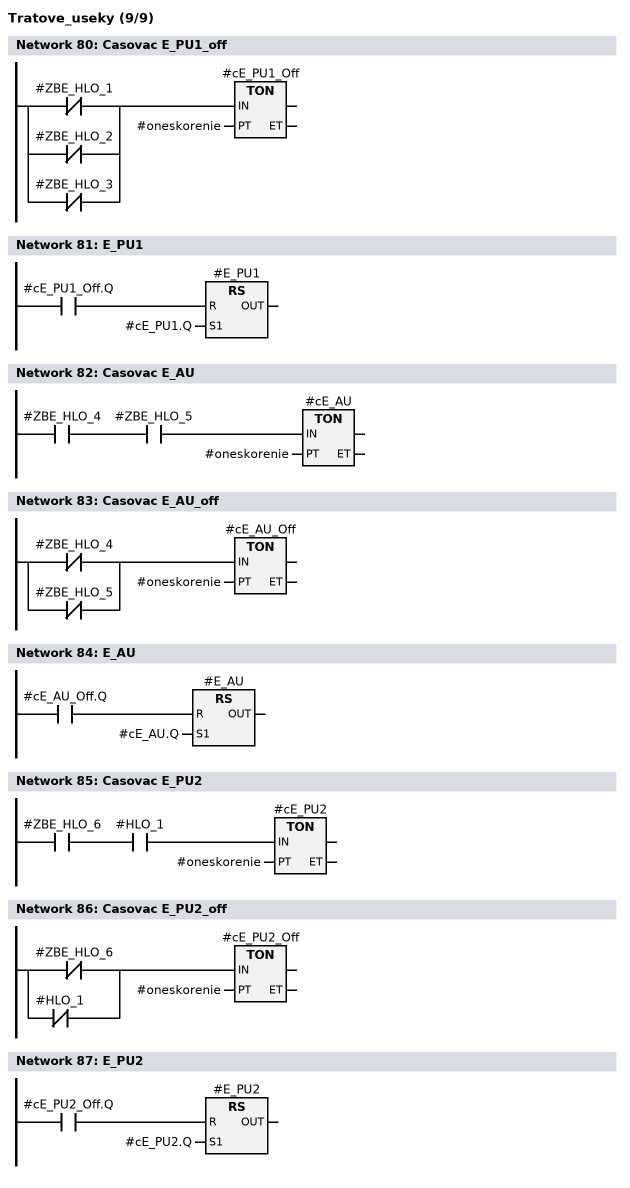
   #cE_PU1_Off.TON(IN := NOT #ZBE_HLO_1 OR NOT #ZBE_HLO_2 OR NOT #ZBE_HLO_3, PT := #oneskorenie);
END_REGION

REGION Network 81: E_PU1
   RUNG wire#powerrail
      Contact( #cE_PU1_Off.Q )
      S_RS(operand := #E_PU1, s1 := #cE_PU1.Q)
   END_RUNG
   // the same network as SCL:
   IF #cE_PU1_Off.Q THEN
       #E_PU1 := FALSE;   // RS flip-flop
   END_IF;
   IF #cE_PU1.Q THEN #E_PU1 := TRUE; END_IF;
END_REGION

REGION Network 82: Casovac E_AU
   #cE_AU.TON(IN := #ZBE_HLO_4 AND #ZBE_HLO_5, PT := #oneskorenie);
END_REGION

REGION Network 83: Casovac E_AU_off
   #cE_AU_Off.TON(IN := NOT #ZBE_HLO_4 OR NOT #ZBE_HLO_5, PT := #oneskorenie);
END_REGION

REGION Network 84: E_AU
   RUNG wire#powerrail
      Contact( #cE_AU_Off.Q )
      S_RS(operand := #E_AU, s1 := #cE_AU.Q)
   END_RUNG
   // the same network as SCL:
   IF #cE_AU_Off.Q THEN
       #E_AU := FALSE;   // RS flip-flop
   END_IF;
   IF #cE_AU.Q THEN #E_AU := TRUE; END_IF;
END_REGION

REGION Network 85: Casovac E_PU2
   #cE_PU2.TON(IN := #ZBE_HLO_6 AND #HLO_1, PT := #oneskorenie);
END_REGION

REGION Network 86: Casovac E_PU2_off
   #cE_PU2_Off.TON(IN := NOT #ZBE_HLO_6 OR NOT #HLO_1, PT := #oneskorenie);
END_REGION

REGION Network 87: E_PU2
   RUNG wire#powerrail
      Contact( #cE_PU2_Off.Q )
      S_RS(operand := #E_PU2, s1 := #cE_PU2.Q)
   END_RUNG
   // the same network as SCL:
   IF #cE_PU2_Off.Q THEN
       #E_PU2 := FALSE;   // RS flip-flop
   END_IF;
   IF #cE_PU2.Q THEN #E_PU2 := TRUE; END_IF;
END_REGION
END_FUNCTION_BLOCK

ORGANIZATION_BLOCK "Main"   // OB1, LAD
TITLE = "Main Program Sweep (Cycle)"
{ S7_Optimized_Access := 'FALSE' }
VERSION : 0.1
   VAR_TEMP
      OB1_EV_CLASS : Byte;   // Bits 0-3 = 1 (Coming event), Bits 4-7 = 1 (Event class 1)
      OB1_SCAN_1 : Byte;   // 1 (Cold restart scan 1 of OB 1), 3 (Scan 2-n of OB 1)
      OB1_PRIORITY : Byte;   // Priority of OB Execution
      OB1_OB_NUMBR : Byte;   // 1 (Organization block 1, OB1)
      OB1_RESERVED_1 : Byte;   // Reserved for system
      OB1_RESERVED_2 : Byte;   // Reserved for system
      OB1_PREV_CYCLE : Int;   // Cycle time of previous OB1 scan (milliseconds)
      OB1_MIN_CYCLE : Int;   // Minimum cycle time of OB1 (milliseconds)
      OB1_MAX_CYCLE : Int;   // Maximum cycle time of OB1 (milliseconds)
      OB1_DATE_TIME : Date_And_Time;   // Date and time OB1 started
   END_VAR
BEGIN

REGION Network 1
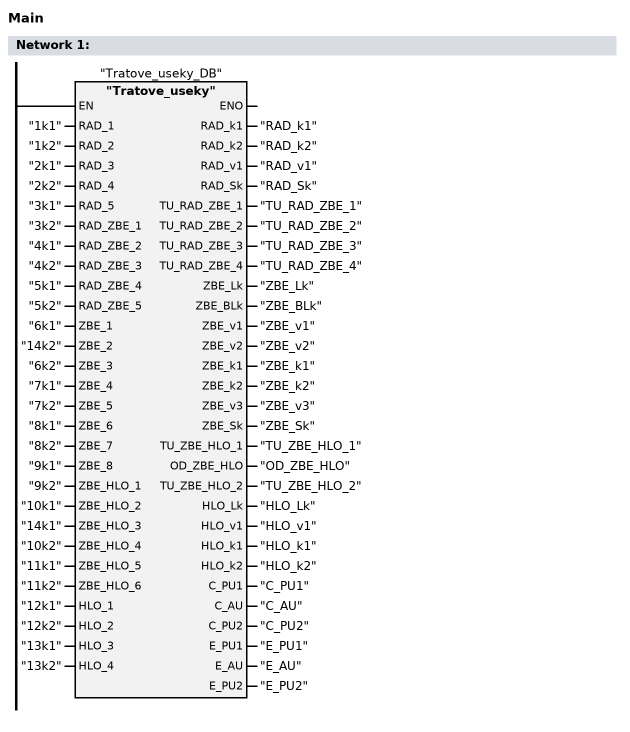
   RUNG wire#powerrail
      "Tratove_useky_DB"(RAD_1 := "1k1", RAD_2 := "1k2", RAD_3 := "2k1", RAD_4 := "2k2", RAD_5 := "3k1", RAD_ZBE_1 := "3k2", RAD_ZBE_2 := "4k1", RAD_ZBE_3 := "4k2", RAD_ZBE_4 := "5k1", RAD_ZBE_5 := "5k2", ZBE_1 := "6k1", ZBE_2 := "14k2", ZBE_3 := "6k2", ZBE_4 := "7k1", ZBE_5 := "7k2", ZBE_6 := "8k1", ZBE_7 := "8k2", ZBE_8 := "9k1", ZBE_HLO_1 := "9k2", ZBE_HLO_2 := "10k1", ZBE_HLO_3 := "14k1", ZBE_HLO_4 := "10k2", ZBE_HLO_5 := "11k1", ZBE_HLO_6 := "11k2", HLO_1 := "12k1", HLO_2 := "12k2", HLO_3 := "13k1", HLO_4 := "13k2", RAD_k1 => "RAD_k1", RAD_k2 => "RAD_k2", RAD_v1 => "RAD_v1", RAD_Sk => "RAD_Sk", TU_RAD_ZBE_1 => "TU_RAD_ZBE_1", TU_RAD_ZBE_2 => "TU_RAD_ZBE_2", TU_RAD_ZBE_3 => "TU_RAD_ZBE_3", TU_RAD_ZBE_4 => "TU_RAD_ZBE_4", ZBE_Lk => "ZBE_Lk", ZBE_BLk => "ZBE_BLk", ZBE_v1 => "ZBE_v1", ZBE_v2 => "ZBE_v2", ZBE_k1 => "ZBE_k1", ZBE_k2 => "ZBE_k2", ZBE_v3 => "ZBE_v3", ZBE_Sk => "ZBE_Sk", TU_ZBE_HLO_1 => "TU_ZBE_HLO_1", OD_ZBE_HLO => "OD_ZBE_HLO", TU_ZBE_HLO_2 => "TU_ZBE_HLO_2", HLO_Lk => "HLO_Lk", HLO_v1 => "HLO_v1", HLO_k1 => "HLO_k1", HLO_k2 => "HLO_k2", C_PU1 => "C_PU1", C_AU => "C_AU", C_PU2 => "C_PU2", E_PU1 => "E_PU1", E_AU => "E_AU", E_PU2 => "E_PU2")
   END_RUNG
   // the same network as SCL:
   "Tratove_useky_DB"(RAD_1 := "1k1",   // "Tratove_useky"
                      RAD_2 := "1k2",
                      RAD_3 := "2k1",
                      RAD_4 := "2k2",
                      RAD_5 := "3k1",
                      RAD_ZBE_1 := "3k2",
                      RAD_ZBE_2 := "4k1",
                      RAD_ZBE_3 := "4k2",
                      RAD_ZBE_4 := "5k1",
                      RAD_ZBE_5 := "5k2",
                      ZBE_1 := "6k1",
                      ZBE_2 := "14k2",
                      ZBE_3 := "6k2",
                      ZBE_4 := "7k1",
                      ZBE_5 := "7k2",
                      ZBE_6 := "8k1",
                      ZBE_7 := "8k2",
                      ZBE_8 := "9k1",
                      ZBE_HLO_1 := "9k2",
                      ZBE_HLO_2 := "10k1",
                      ZBE_HLO_3 := "14k1",
                      ZBE_HLO_4 := "10k2",
                      ZBE_HLO_5 := "11k1",
                      ZBE_HLO_6 := "11k2",
                      HLO_1 := "12k1",
                      HLO_2 := "12k2",
                      HLO_3 := "13k1",
                      HLO_4 := "13k2",
                      RAD_k1 => "RAD_k1",
                      RAD_k2 => "RAD_k2",
                      RAD_v1 => "RAD_v1",
                      RAD_Sk => "RAD_Sk",
                      TU_RAD_ZBE_1 => "TU_RAD_ZBE_1",
                      TU_RAD_ZBE_2 => "TU_RAD_ZBE_2",
                      TU_RAD_ZBE_3 => "TU_RAD_ZBE_3",
                      TU_RAD_ZBE_4 => "TU_RAD_ZBE_4",
                      ZBE_Lk => "ZBE_Lk",
                      ZBE_BLk => "ZBE_BLk",
                      ZBE_v1 => "ZBE_v1",
                      ZBE_v2 => "ZBE_v2",
                      ZBE_k1 => "ZBE_k1",
                      ZBE_k2 => "ZBE_k2",
                      ZBE_v3 => "ZBE_v3",
                      ZBE_Sk => "ZBE_Sk",
                      TU_ZBE_HLO_1 => "TU_ZBE_HLO_1",
                      OD_ZBE_HLO => "OD_ZBE_HLO",
                      TU_ZBE_HLO_2 => "TU_ZBE_HLO_2",
                      HLO_Lk => "HLO_Lk",
                      HLO_v1 => "HLO_v1",
                      HLO_k1 => "HLO_k1",
                      HLO_k2 => "HLO_k2",
                      C_PU1 => "C_PU1",
                      C_AU => "C_AU",
                      C_PU2 => "C_PU2",
                      E_PU1 => "E_PU1",
                      E_AU => "E_AU",
                      E_PU2 => "E_PU2");
END_REGION
END_ORGANIZATION_BLOCK

// ===== PLC "PLC_1"  CPU 1214C DC/DC/DC =====

VAR_GLOBAL   // PLC tag table "Default tag table"
   "Clock_Byte" AT %MB100 : Byte;
   "Clock_10Hz" AT %M100.0 : Bool;
   "Clock_5Hz" AT %M100.1 : Bool;
   "Clock_2.5Hz" AT %M100.2 : Bool;
   "Clock_2Hz" AT %M100.3 : Bool;
   "Clock_1.25Hz" AT %M100.4 : Bool;
   "Clock_1Hz" AT %M100.5 : Bool;
   "Clock_0.625Hz" AT %M100.6 : Bool;
   "Clock_0.5Hz" AT %M100.7 : Bool;
   "TEST" AT %Q16.0 : Bool;
END_VAR

VAR_GLOBAL   // PLC tag table "C_Memory"
   "C_P_PU_BA" AT %M0.5 : Bool;   // Priecestie C: porucha prib useku-smer BA
   "C_P_AU" AT %M0.4 : Bool;   // Priecestie C: porucha anulovacieho useku
   "C_P_PU_AB" AT %M0.3 : Bool;   // Priecestie C: porucha prib. useku-smer AB
   "C_PU_BA" AT %M0.2 : Bool;   // Priecestie C: priblizovaci usek-smer BA
   "C_AU" AT %M0.1 : Bool;   // Priecestie C: anulovaci usek
   "C_PU_AB" AT %M0.0 : Bool;   // Priecestie C: priblizovaci usek-smer AB
   "C_P_Z_H" AT %M0.6 : Bool;   // Priecestie C: porucha zavory hore
   "C_P_Z_D" AT %M0.7 : Bool;   // Priecestie C: porucha zavory dole
   "C_P_C" AT %M1.0 : Bool;   // Priecestie C: porucha cervenej
   "C_P_B" AT %M1.1 : Bool;   // Priecestie C: porucha bielej
   "C_otvorene" AT %M1.2 : Bool;
   "C_zatvorene" AT %M1.3 : Bool;
   "C_predzvananie" AT %M1.4 : Bool;
   "C_manual_zatvor" AT %M3.2 : Bool;
END_VAR

VAR_GLOBAL   // PLC tag table "C_Výstupy"
   "C_C" AT %Q0.0 : Bool;   // Priecestie C: Cervena
   "C_B" AT %Q0.1 : Bool;   // Priecestie C: Biela
   "C_P" AT %Q0.2 : Bool;   // Priecestie C: Porucha
   "C_Z_H" AT %Q0.3 : Bool;   // Priecestie C: Motor Hore
   "C_Z_D" AT %Q0.4 : Bool;   // Priecestie C: Motor Dole
END_VAR

VAR_GLOBAL   // PLC tag table "E_Výstupy"
   "E_C" AT %Q0.5 : Bool;   // Priecestie E: Cervena
   "E_B" AT %Q0.6 : Bool;   // Priecestie E: Biela
   "E_P" AT %Q0.7 : Bool;   // Priecestie E: Porucha
   "E_Z_H" AT %Q1.0 : Bool;   // Priecestie E: Motor Hore
   "E_Z_D" AT %Q1.1 : Bool;   // Priecestie E: Motor Dole
END_VAR

VAR_GLOBAL   // PLC tag table "E_Memory"
   "E_PU_AB" AT %M2.0 : Bool;   // Priecestie E: priblizovaci usek-smer AB
   "E_AU" AT %M2.1 : Bool;   // Priecestie E: anulovaci usek
   "E_PU_BA" AT %M2.2 : Bool;   // Priecestie E: priblizovaciu usek-smer BA
   "E_P_PU_AB" AT %M2.3 : Bool;   // Priecestie E: porucha prib. useku-smer AB
   "E_P_AU" AT %M2.4 : Bool;   // Priecestie E: porucha anulovacieho useku
   "E_P_PU_BA" AT %M2.5 : Bool;   // Priecestie E: porucha prib. useku-smer BA
   "E_P_Z_H" AT %M2.6 : Bool;   // Priecestie E: porucha zavory hore
   "E_P_Z_D" AT %M2.7 : Bool;   // Priecestie E: porucha zavory dole
   "E_P_C" AT %M3.0 : Bool;   // Priecestie E: porucha cervenej
   "E_P_B" AT %M3.1 : Bool;   // Priecestie E: porucha bielej
   "E_otvorene" AT %M1.5 : Bool;
   "E_zatvorene" AT %M1.6 : Bool;
   "E_predzvananie" AT %M1.7 : Bool;
   "E_manual_zatvor" AT %M3.3 : Bool;
END_VAR

VAR_GLOBAL   // PLC tag table "AB-navestidla"
   "AB-18_ze" AT %Q4.0 : Bool;
   "AB-18_ce" AT %Q4.1 : Bool;
   "AB-18_zl" AT %Q3.7 : Bool;
   "AB-19_ze" AT %Q4.3 : Bool;
   "AB-19_ce" AT %Q4.4 : Bool;
   "AB-19_zl" AT %Q4.2 : Bool;
   "AB-28_ze" AT %Q4.6 : Bool;
   "AB-28_ce" AT %Q4.7 : Bool;
   "AB-28_zl" AT %Q4.5 : Bool;
   "AB-29_ze" AT %Q5.1 : Bool;
   "AB-29_ce" AT %Q5.2 : Bool;
   "AB-29_zl" AT %Q5.0 : Bool;
   "AB-39_ze" AT %Q5.4 : Bool;
   "AB-39_ce" AT %Q5.5 : Bool;
   "AB-39_zl" AT %Q5.3 : Bool;
   "AB-40_ze" AT %Q5.7 : Bool;
   "AB-40_ce" AT %Q6.0 : Bool;
   "AB-40_zl" AT %Q5.6 : Bool;
END_VAR

VAR_GLOBAL   // PLC tag table "AH-navestidla"
   "AH-Lo_ze" AT %Q11.6 : Bool;
   "AH-Lo_ce" AT %Q11.7 : Bool;
   "AH-Lo_bi" AT %Q12.0 : Bool;
   "AH-PrLo_ze" AT %Q11.2 : Bool;
   "AH-PrLo_zl" AT %Q11.3 : Bool;
   "AH-So_ze" AT %Q12.1 : Bool;
   "AH-So_ce" AT %Q12.2 : Bool;
   "AH-So_bi" AT %Q12.3 : Bool;
   "AH-PrSo_ze" AT %Q11.4 : Bool;
   "AH-PrSo_zl" AT %Q11.5 : Bool;
END_VAR

VAR_GLOBAL   // PLC tag table "tratove_useky"
   "RAD_k1" AT %I2.0 : Bool;
   "RAD_k2" AT %I2.1 : Bool;
   "RAD_v1" AT %I2.2 : Bool;
   "RAD_Sk" AT %I2.3 : Bool;
   "RAD_ZBE_TU1" AT %I2.4 : Bool;
   "RAD_ZBE_TU2" AT %I2.5 : Bool;
   "RAD_ZBE_TU3" AT %I2.6 : Bool;
   "RAD_ZBE_TU4" AT %I2.7 : Bool;
   "ZBE_Lk" AT %I3.0 : Bool;
   "ZBE_BLk" AT %I3.1 : Bool;
   "ZBE_v1" AT %I3.2 : Bool;
   "ZBE_v2" AT %I3.3 : Bool;
   "ZBE_k1" AT %I3.4 : Bool;
   "ZBE_k2" AT %I3.5 : Bool;
   "ZBE_v3" AT %I3.6 : Bool;
   "ZBE_Sk" AT %I3.7 : Bool;
   "ZBE_HLO_TU1" AT %I4.6 : Bool;
   "ZBE_HLO_TU2" AT %I4.7 : Bool;
   "HLO_Lk" AT %I5.0 : Bool;
   "HLO_v1" AT %I5.1 : Bool;
   "HLO_k1" AT %I5.2 : Bool;
   "HLO_k2" AT %I5.3 : Bool;
   "Priec_C_PU1" AT %I4.0 : Bool;
   "Priec_C_AU" AT %I4.1 : Bool;
   "Priec_C_PU2" AT %I4.2 : Bool;
   "Priec_E_PU1" AT %I4.3 : Bool;
   "Priec_E_AU" AT %I4.4 : Bool;
   "Priec_E_PU2" AT %I4.5 : Bool;
   "ZBE_HLO_OD" AT %I5.4 : Bool;
END_VAR

VAR_GLOBAL   // PLC tag table "St-RAD_navestidla"
   "RAD_L1_zl" AT %Q2.0 : Bool;
   "RAD_L1_ze" AT %Q2.1 : Bool;
   "RAD_L1_ce" AT %Q2.2 : Bool;
   "RAD_L1_bi" AT %Q2.3 : Bool;
   "RAD_L2_zl_h" AT %Q2.4 : Bool;
   "RAD_L2_ze" AT %Q2.5 : Bool;
   "RAD_L2_ce" AT %Q2.6 : Bool;
   "RAD_L2_bi" AT %Q2.7 : Bool;
   "RAD_L2_zl_d" AT %Q3.0 : Bool;
   "RAD_S_zl_h" AT %Q3.3 : Bool;
   "RAD_S_ce" AT %Q3.4 : Bool;
   "RAD_S_bi" AT %Q3.5 : Bool;
   "RAD_S_zl_d" AT %Q3.6 : Bool;
   "RAD_Se1_bi" AT %Q3.1 : Bool;
   "RAD_Se1_mo" AT %Q3.2 : Bool;
   "RAD_stav_L1" AT %MB8 : Byte;
   "RAD_stav_L2" AT %MB9 : Byte;
   "Rad_stav_S" AT %MB10 : Byte;
   "Rad_stav_Se1" AT %MB11 : Byte;
END_VAR

VAR_GLOBAL   // PLC tag table "St-ZBE_navestidla"
   "ZBE_L_zl_h" AT %Q6.1 : Bool;
   "ZBE_L_ze" AT %Q6.2 : Bool;
   "ZBE_L_ce" AT %Q6.3 : Bool;
   "ZBE_L_bi" AT %Q6.4 : Bool;
   "ZBE_L_zl_d" AT %Q6.5 : Bool;
   "ZBE_S1_zl_h" AT %Q7.2 : Bool;
   "ZBE_S1_ze" AT %Q7.3 : Bool;
   "ZBE_S1_ce" AT %Q7.4 : Bool;
   "ZBE_S1_bi" AT %Q7.5 : Bool;
   "ZBE_S2_zl_h" AT %Q7.6 : Bool;
   "ZBE_S2_ze" AT %Q7.7 : Bool;
   "ZBE_S2_ce" AT %Q8.0 : Bool;
   "ZBE_S2_bi" AT %Q8.1 : Bool;
   "ZBE_S2_zl_d" AT %Q8.2 : Bool;
   "ZBE_L1_ze" AT %Q8.3 : Bool;
   "ZBE_L1_ce" AT %Q8.4 : Bool;
   "ZBE_L1_bi" AT %Q8.5 : Bool;
   "ZBE_L2_ze" AT %Q8.6 : Bool;
   "ZBE_L2_ce" AT %Q8.7 : Bool;
   "ZBE_L2_bi" AT %Q9.0 : Bool;
   "ZBE_L2_zl_d" AT %Q9.1 : Bool;
   "ZBE_S_zl_h" AT %Q9.4 : Bool;
   "ZBE_S_ze" AT %Q9.5 : Bool;
   "ZBE_S_ce" AT %Q9.6 : Bool;
   "ZBE_S_bi" AT %Q9.7 : Bool;
   "ZBE_S_zl_d" AT %Q10.0 : Bool;
   "ZBE_Se1_bi" AT %Q6.6 : Bool;
   "ZBE_Se1_mo" AT %Q6.7 : Bool;
   "ZBE_Se2_bi" AT %Q7.0 : Bool;
   "ZBE_Se2_mo" AT %Q7.1 : Bool;
   "ZBE_Se3_bi" AT %Q9.2 : Bool;
   "ZBE_Se3_mo" AT %Q9.3 : Bool;
   "ZBE_PrS_zl" AT %Q10.1 : Bool;
   "ZBE_PrS_ze" AT %Q10.2 : Bool;
   "ZBE_BL_zl_h" AT %Q10.3 : Bool;
   "ZBE_BL_ze" AT %Q10.4 : Bool;
   "ZBE_BL_ce" AT %Q10.5 : Bool;
   "ZBE_BL_bi" AT %Q10.6 : Bool;
   "ZBE_BL_zl_d" AT %Q10.7 : Bool;
   "ZBE_PrBL_zl" AT %Q11.0 : Bool;
   "ZBE_PrBL_ze" AT %Q11.1 : Bool;
   "ZBE_stav_L" AT %MB12 : Byte;
   "ZBE_stav_BL" AT %MB13 : Byte;
   "ZBE_stav_S" AT %MB14 : Byte;
   "ZBE_stav_L1" AT %MB15 : Byte;
   "ZBE_svtav_L2" AT %MB16 : Byte;
   "ZBE_stav_S1" AT %MB17 : Byte;
   "ZBE_stav_S2" AT %MB18 : Byte;
   "ZBE_stav_Se1" AT %MB19 : Byte;
   "ZBE_stav_Se2" AT %MB20 : Byte;
   "ZBE_stav_Se3" AT %MB21 : Byte;
   "ZBE_OD_k1-RAD" AT %M6.0 : Bool;   // Ochranna draha k1 od Radosiny
   "ZBE_OD_k1-HLO" AT %M6.1 : Bool;   // Ochranna draha k1 od Hlohovca
   "ZBE_OD_k2-LUZ" AT %M6.2 : Bool;   // Ochranna draha k2 od Luzianok
   "ZBE_So_navMan" AT %MB28 : Byte;
END_VAR

VAR_GLOBAL   // PLC tag table "St-HLO_navestidla"
   "HLO_PrL_zl" AT %Q12.4 : Bool;
   "HLO_PrL_ze" AT %Q12.5 : Bool;
   "HLO_L_zl_h" AT %Q12.6 : Bool;
   "HLO_L_ce" AT %Q12.7 : Bool;
   "HLO_L_bi" AT %Q13.0 : Bool;
   "HLO_L_zl_d" AT %Q13.1 : Bool;
   "HLO_S1_ze" AT %Q13.4 : Bool;
   "HLO_S1_ce" AT %Q13.5 : Bool;
   "HLO_S1_bi" AT %Q13.6 : Bool;
   "HLO_S2_ze" AT %Q13.7 : Bool;
   "HLO_S2_ce" AT %Q14.0 : Bool;
   "HLO_S2_bi" AT %Q14.1 : Bool;
   "HLO_S2_zl_d" AT %Q14.2 : Bool;
   "HLO_Se1_bi" AT %Q13.3 : Bool;
   "HLO_Se1_mo" AT %Q13.2 : Bool;
   "HLO_stav_L" AT %MB22 : Byte;
   "HLO_stav_S1" AT %MB23 : Byte;
   "HLO_stav_S2" AT %MB24 : Byte;
   "HLO_stav_Se1" AT %MB25 : Byte;
   "HLO_Lo_navMan" AT %MB27 : Byte;
END_VAR

VAR_GLOBAL   // PLC tag table "vyhybky"
   "RAD_vyh1O" AT %Q15.0 : Bool;
   "ZBE_vyh1O" AT %Q15.1 : Bool;
   "ZBE_vyh2O" AT %Q15.2 : Bool;
   "ZBE_vyh3O" AT %Q15.3 : Bool;
   "HLO_vyh1O" AT %Q15.4 : Bool;
   "RAD_vyh1IP" AT %I0.0 : Bool;
   "RAD_vyh1IM" AT %I0.1 : Bool;
   "ZBE_vyh1IP" AT %I0.2 : Bool;
   "ZBE_vyh1IM" AT %I0.3 : Bool;
   "ZBE_vyh2IP" AT %I0.4 : Bool;
   "ZBE_Vyh2IM" AT %I0.5 : Bool;
   "ZBE_vyh3IP" AT %I0.6 : Bool;
   "ZBE_vyh3IM" AT %I0.7 : Bool;
   "HLO_vyh1IP" AT %I1.0 : Bool;
   "HLO_vyh1IM" AT %I1.1 : Bool;
   "ZBE_1-2prestP" AT %M4.2 : Bool;   // Zbe V1-V2: prestavovanie do plusu
   "ZBE_3prestP" AT %M4.4 : Bool;   // Zbe V3: prestavovanie do plusu
   "HLO_1prestP" AT %M4.6 : Bool;   // Hlo V1: prestavovanie do plusu
   "RAD_1prestM" AT %M4.1 : Bool;   // Rad V1: prestavovanie do minusu
   "ZBE_1-2prestM" AT %M4.3 : Bool;   // Zbe V1-V2: prestavovanie do minusu
   "ZBE_3prestM" AT %M4.5 : Bool;   // Zbe V3: prestavovanie do minusu
   "HLO_1prestM" AT %M4.7 : Bool;   // Hlo V1: prestavovanie do minusu
   "RAD_1_smer" AT %M5.0 : Bool;   // Rad V1: smer
   "ZBE_1_smer" AT %M5.4 : Bool;   // Zbe V1: smer
   "ZBE_2_smer" AT %M5.5 : Bool;   // Zbe V2: smer
   "ZBE_3_smer" AT %M5.2 : Bool;   // Zbe V3: smer
   "HLO_1_smer" AT %M5.3 : Bool;   // Hlo V1: smer
   "RAD_1prestP" AT %M4.0 : Bool;   // Rad V1: prestavovanie do plusu
   "ZBE_1-2_smer" AT %M5.1 : Bool;   // Zbe V1-2: smer
   "ZBE_1_prestP" AT %M5.6 : Bool;   // Zbe V1: prestavovanie do plusu
   "ZBE_1_prestM" AT %M5.7 : Bool;   // Zbe V1: prestavovanie do minusu
   "ZBE_2_prestP" AT %M6.3 : Bool;   // Zbe V2: prestavovanie do plusu
   "ZBE_2_prestM" AT %M6.4 : Bool;   // Zbe V2: prestavovanie do minusu
END_VAR

VAR_GLOBAL   // PLC tag table "TS"
   "smer_TS_RAD-ZBE" AT %M7.0 : Bool;   // smer tratoveho suhlasu (0->lichy, 1->sudy)
   "smer_TS_ZBE-HLO" AT %M7.1 : Bool;   // smer tratoveho suhlasu (0->lichy, 1->sudy)
   "volnost_MU_Rad-Zbe" AT %M7.3 : Bool;   // volnost medzist useku RAD - ZBE
   "volnost_MU_Zbe_AH" AT %M7.4 : Bool;   // volnost medzist useku ZBE - AH
   "odchod_RAD" AT %M26.0 : Bool;
   "odchod_ZBE-R" AT %M26.1 : Bool;
   "odchod_ZBE-H" AT %M26.3 : Bool;
   "odchodHLO" AT %M26.4 : Bool;
   "predhlaska_ZBE" AT %M29.0 : Bool;
   "predhlaska_HLO" AT %M29.1 : Bool;
   "odhlaska_ZBE" AT %M29.4 : Bool;
   "odhlaska_HLO" AT %M29.5 : Bool;
   "predhlaska_Lo" AT %M29.2 : Bool;
   "predhlaska_So" AT %M29.3 : Bool;
   "odhlaska_Lo" AT %M29.6 : Bool;
   "odhlaska_So" AT %M29.7 : Bool;
   "volnost_MU_Hlo_AH" AT %M7.5 : Bool;   // volnost medzist useku HLO - AH
END_VAR

DATA_BLOCK "Automaticke_hradlo_Lo"   // DB1
{ S7_Optimized_Access := 'TRUE' }
VERSION : 0.1
// stored: InstanceOfName Automaticke_hradlo
"Automaticke_hradlo"
BEGIN
END_DATA_BLOCK

DATA_BLOCK "Automaticke_hradlo_So"   // DB2
{ S7_Optimized_Access := 'TRUE' }
VERSION : 0.1
// stored: InstanceOfName Automaticke_hradlo
"Automaticke_hradlo"
BEGIN
END_DATA_BLOCK

DATA_BLOCK "Radosina_DB"   // DB3
{ S7_Optimized_Access := 'TRUE' }
VERSION : 0.1
// stored: InstanceOfName Radosina
"Radosina"
BEGIN
END_DATA_BLOCK

DATA_BLOCK "Zbehy_DB"   // DB4
{ S7_Optimized_Access := 'TRUE' }
VERSION : 0.1
// stored: InstanceOfName Zbehy
"Zbehy"
BEGIN
END_DATA_BLOCK

DATA_BLOCK "Hlohovec_DB"   // DB5
{ S7_Optimized_Access := 'TRUE' }
VERSION : 0.1
// stored: InstanceOfName Hlohovec
"Hlohovec"
BEGIN
END_DATA_BLOCK

DATA_BLOCK "Autoblok_18"   // DB6
{ S7_Optimized_Access := 'TRUE' }
VERSION : 0.1
// stored: InstanceOfName Autoblok
"Autoblok"
BEGIN
END_DATA_BLOCK

DATA_BLOCK "Autoblok_19"   // DB7
{ S7_Optimized_Access := 'TRUE' }
VERSION : 0.1
// stored: InstanceOfName Autoblok
"Autoblok"
BEGIN
END_DATA_BLOCK

DATA_BLOCK "Autoblok_28"   // DB8
{ S7_Optimized_Access := 'TRUE' }
VERSION : 0.1
// stored: InstanceOfName Autoblok
"Autoblok"
BEGIN
END_DATA_BLOCK

DATA_BLOCK "Autoblok_29"   // DB9
{ S7_Optimized_Access := 'TRUE' }
VERSION : 0.1
// stored: InstanceOfName Autoblok
"Autoblok"
BEGIN
END_DATA_BLOCK

DATA_BLOCK "Autoblok_40"   // DB10
{ S7_Optimized_Access := 'TRUE' }
VERSION : 0.1
// stored: InstanceOfName Autoblok
"Autoblok"
BEGIN
END_DATA_BLOCK

DATA_BLOCK "Autoblok_39"   // DB11
{ S7_Optimized_Access := 'TRUE' }
VERSION : 0.1
// stored: InstanceOfName Autoblok
"Autoblok"
BEGIN
END_DATA_BLOCK

DATA_BLOCK "Výhybka_RAD1"   // DB12
{ S7_Optimized_Access := 'TRUE' }
VERSION : 0.1
// stored: InstanceOfName Vyhybka
"Vyhybka"
BEGIN
END_DATA_BLOCK

DATA_BLOCK "Výhybka_ZBE1"   // DB13
{ S7_Optimized_Access := 'TRUE' }
VERSION : 0.1
// stored: InstanceOfName Vyhybka
"Vyhybka"
BEGIN
END_DATA_BLOCK

DATA_BLOCK "Výhybka_ZBE2"   // DB14
{ S7_Optimized_Access := 'TRUE' }
VERSION : 0.1
// stored: InstanceOfName Vyhybka
"Vyhybka"
BEGIN
END_DATA_BLOCK

DATA_BLOCK "Výhybka_ZBE3"   // DB15
{ S7_Optimized_Access := 'TRUE' }
VERSION : 0.1
// stored: InstanceOfName Vyhybka
"Vyhybka"
BEGIN
END_DATA_BLOCK

DATA_BLOCK "Výhybka_HLO1"   // DB16
{ S7_Optimized_Access := 'TRUE' }
VERSION : 0.1
// stored: InstanceOfName Vyhybka
"Vyhybka"
BEGIN
END_DATA_BLOCK

DATA_BLOCK "Config"   // DB17
{ S7_Optimized_Access := 'TRUE' }
VERSION : 0.1
   VAR
      Dly_C_PU_AB : Time := T#600ms;   // Oneskorenie v priblizovacom useku AB (C)
      Dly_C_AU : Time := T#600ms;   // Oneskorenie v anulovacom useku (C)
      Dly_C_PU_BA : Time := T#600ms;   // Oneskorenie v priblizovacom useku BA (C)
      AC_C : Time := T#20s;   // Cas anulacie (C)
      VSC_C : Time := T#2500ms;   // Vystrazny sklapaci cas (C)
      ZC_C : Time := T#2500ms;   // Oneskorenie vypnutia svetelnej vysrahy (C)
      Dly_E_PU_AB : Time := T#600ms;   // Oneskorenie v priblizovacom useku AB (E)
      Dly_E_AU : Time := T#600ms;   // Oneskorenie v anulovacom useku (E)
      Dly_E_PU_BA : Time := T#600ms;   // Oneskorenie v priblizovacom useku BA (E)
      AC_E : Time := T#20s;   // Cas anulacie (E)
      VSC_E : Time := T#2500ms;   // Vystrazny sklapaci cas (E)
      ZC_E : Time := T#2500ms;   // Oneskorenie vypnutia svetelnej vystrahy (E)
   END_VAR
BEGIN
END_DATA_BLOCK

DATA_BLOCK "Priecestie_C_DB"   // DB18
{ S7_Optimized_Access := 'TRUE' }
VERSION : 0.1
// stored: InstanceOfName Priecestie
"Priecestie"
BEGIN
END_DATA_BLOCK

DATA_BLOCK "Priecestie_E_DB"   // DB19
{ S7_Optimized_Access := 'TRUE' }
VERSION : 0.1
// stored: InstanceOfName Priecestie
"Priecestie"
BEGIN
END_DATA_BLOCK

FUNCTION_BLOCK "Automaticke_hradlo"   // FB1, LAD
{ S7_Optimized_Access := 'TRUE' }
VERSION : 0.1
   VAR_INPUT
      TS : Bool;
      smerNav : Bool;   // 0-lichy, 1-sudy
      usek_za_nav : Bool;
      usek_pred_nav : Bool;
      navMan : Byte;
      blikac : Bool;
   END_VAR
   VAR_OUTPUT
      zelena : Bool;
      cervena : Bool;
      biela : Bool;
      Pr_zelena : Bool;
      Pr_zlta : Bool;
   END_VAR
   VAR_IN_OUT
      dosla_predhlaska : Bool;
      dosla_odhlaska : Bool;
      odoslana_predhlaska : Bool;
      odoslana_odhlaska : Bool := true;
   END_VAR
   VAR
      stav : Byte;
   END_VAR
   VAR_TEMP   // added for the SCL form of the ladder/FBD networks
      _w1 : Bool;
   END_VAR
BEGIN

REGION Network 1: Zakladny stav
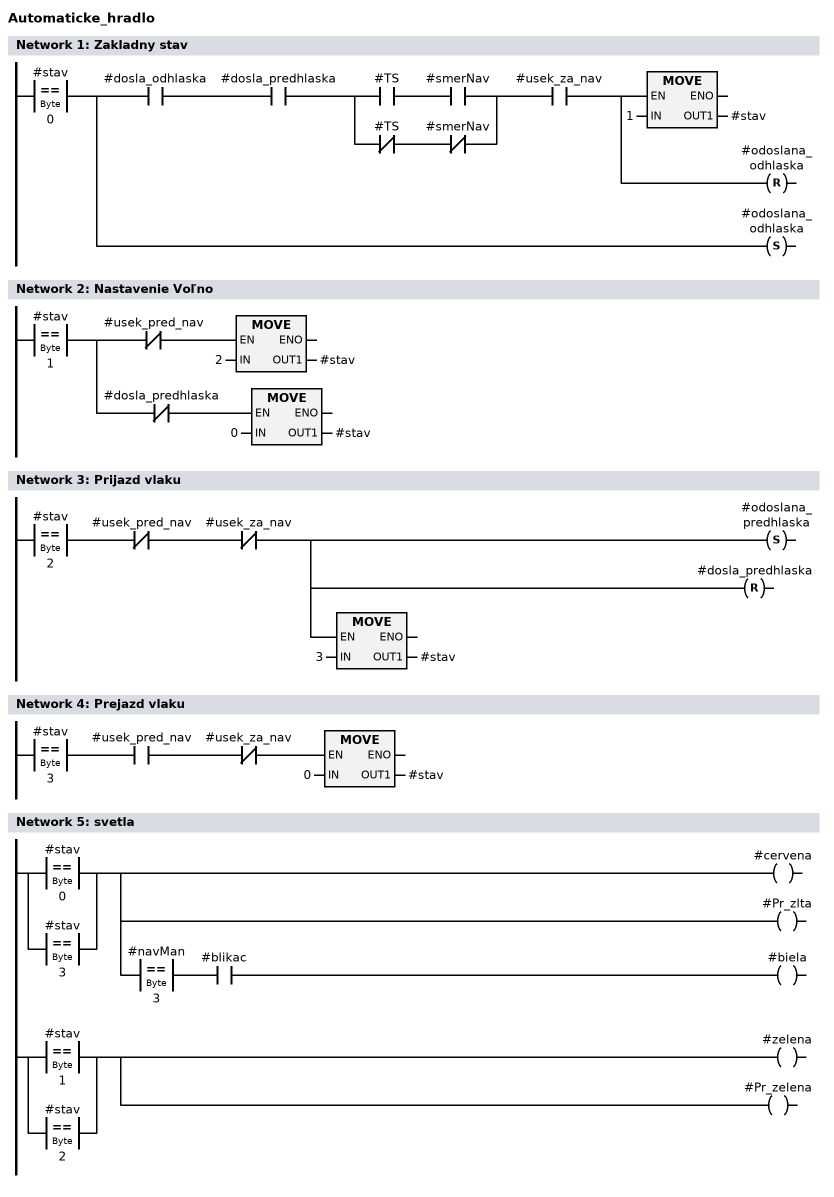
   RUNG wire#powerrail
      { S7_Templates := "SrcType := Byte" } EQ_Contact(in1 := #stav, in2 := 0)
      wire#w1
      Contact( #dosla_odhlaska )
      Contact( #dosla_predhlaska )
      wire#w2
      Contact( #TS )
      Contact( #smerNav )
      wire#w3
      Contact( #usek_za_nav )
      wire#w4
      { S7_GenerateENO := "TRUE" } Move(in := 1, out1 => #stav)
   END_RUNG
   RUNG wire#w2
      I_Contact( #TS )
      I_Contact( #smerNav )
   END_RUNG wire#w3
   RUNG wire#w4
      R_Coil( #odoslana_odhlaska )
   END_RUNG
   RUNG wire#w1
      S_Coil( #odoslana_odhlaska )
   END_RUNG
   // the same network as SCL:
   #_w1 := #stav = 0;
   IF #_w1 AND #dosla_odhlaska AND #dosla_predhlaska AND ((#TS AND #smerNav) OR (NOT #TS AND NOT #smerNav)) AND #usek_za_nav THEN
       #stav := 1;
       #odoslana_odhlaska := FALSE;
   END_IF;
   IF #_w1 THEN #odoslana_odhlaska := TRUE; END_IF;
END_REGION

REGION Network 2: Nastavenie Voľno
   RUNG wire#powerrail
      { S7_Templates := "SrcType := Byte" } EQ_Contact(in1 := #stav, in2 := 1)
      wire#w1
      I_Contact( #usek_pred_nav )
      { S7_GenerateENO := "TRUE" } Move(in := 2, out1 => #stav)
   END_RUNG
   RUNG wire#w1
      I_Contact( #dosla_predhlaska )
      { S7_GenerateENO := "TRUE" } Move(in := 0, out1 => #stav)
   END_RUNG
   // the same network as SCL:
   #_w1 := #stav = 1;
   IF #_w1 AND NOT #usek_pred_nav THEN #stav := 2; END_IF;
   IF #_w1 AND NOT #dosla_predhlaska THEN #stav := 0; END_IF;
END_REGION

REGION Network 3: Prijazd vlaku
   RUNG wire#powerrail
      { S7_Templates := "SrcType := Byte" } EQ_Contact(in1 := #stav, in2 := 2)
      I_Contact( #usek_pred_nav )
      I_Contact( #usek_za_nav )
      wire#w1
      S_Coil( #odoslana_predhlaska )
   END_RUNG
   RUNG wire#w1
      R_Coil( #dosla_predhlaska )
   END_RUNG
   RUNG wire#w1
      { S7_GenerateENO := "TRUE" } Move(in := 3, out1 => #stav)
   END_RUNG
   // the same network as SCL:
   IF (#stav = 2) AND NOT #usek_pred_nav AND NOT #usek_za_nav THEN
       #odoslana_predhlaska := TRUE;
       #dosla_predhlaska := FALSE;
       #stav := 3;
   END_IF;
END_REGION

REGION Network 4: Prejazd vlaku
   RUNG wire#powerrail
      { S7_Templates := "SrcType := Byte" } EQ_Contact(in1 := #stav, in2 := 3)
      Contact( #usek_pred_nav )
      I_Contact( #usek_za_nav )
      { S7_GenerateENO := "TRUE" } Move(in := 0, out1 => #stav)
   END_RUNG
   // the same network as SCL:
   IF (#stav = 3) AND #usek_pred_nav AND NOT #usek_za_nav THEN #stav := 0; END_IF;
END_REGION

REGION Network 5: svetla
   RUNG wire#powerrail
      { S7_Templates := "SrcType := Byte" } EQ_Contact(in1 := #stav, in2 := 0)
      wire#w1
      Coil( #cervena )
   END_RUNG
   RUNG wire#powerrail
      { S7_Templates := "SrcType := Byte" } EQ_Contact(in1 := #stav, in2 := 3)
   END_RUNG wire#w1
   RUNG wire#w1
      Coil( #Pr_zlta )
   END_RUNG
   RUNG wire#w1
      { S7_Templates := "SrcType := Byte" } EQ_Contact(in1 := #navMan, in2 := 3)
      Contact( #blikac )
      Coil( #biela )
   END_RUNG
   RUNG wire#powerrail
      { S7_Templates := "SrcType := Byte" } EQ_Contact(in1 := #stav, in2 := 1)
      wire#w2
      Coil( #zelena )
   END_RUNG
   RUNG wire#powerrail
      { S7_Templates := "SrcType := Byte" } EQ_Contact(in1 := #stav, in2 := 2)
   END_RUNG wire#w2
   RUNG wire#w2
      Coil( #Pr_zelena )
   END_RUNG
   // the same network as SCL:
   #cervena := (#stav = 0) OR (#stav = 3);
   #Pr_zlta := #cervena;
   #biela := #cervena AND (#navMan = 3) AND #blikac;
   #zelena := (#stav = 1) OR (#stav = 2);
   #Pr_zelena := #zelena;
END_REGION
END_FUNCTION_BLOCK

FUNCTION_BLOCK "Priecestie"   // FB2, LAD
{ S7_Optimized_Access := 'TRUE' }
VERSION : 0.1
   VAR_INPUT
      PU_AB : Bool;   // Priblizovaci usek-smer AB
      AU : Bool;   // Anulovaci usek
      PU_BA : Bool;   // Priblizovaci usek-smer BA
      P_Z_H : Bool;   // Porucha zavora hore
      P_Z_D : Bool;   // Porucha zavora dole
      AC : Time;   // Anulovaci cas
      VSC : Time;   // Vystrazny sklapaci cas
      ZC : Time;
      manual : Bool;
   END_VAR
   VAR_OUTPUT
      Z_H : Bool;   // Zavora hore
      Z_D : Bool;   // Zavora dole
      C : Bool;   // Cervena
      "B" : Bool;   // Biela
      predzvananie : Bool;
      priecestie_zatvorene : Bool;
      priecestie_otvorene : Bool;
   END_VAR
   VAR
      S_AB : Bool;   // Smer A->B
      S_BA : Bool;   // Smer B->A
      Vystraha : Bool;   // Spustenie vystrahy
      R_AB : Bool;   // Ukoncenie vystrahy pre smer A->B
      R_BA : Bool;   // Ukoncenie vystrahy pre smer B->A
      R_BBA : Bool;   // Reset vystrahy bez prejazdu priecestia smerom BA
      R_BAB : Bool;   // Reset vystrahy bez prejazdu priecestia smerom AB
      P1 : Bool;   // Pomocna premenna pre otvorenie zavor
      P2 : Bool;   // Pomocna premenna
      P3 : Bool;   // Pomocna premenna
      CA_time : Time;   // Cas anulacie
      CA : TON_TIME;   // Zaznamenanie casu anulacie
      SmerDB : "Detekcia_Smeru_Jazdy";   // Detekcia smeru jazdy KV
      TON1 : TON_TIME;   // Vystrazny sklapaci cas
      TOF1 : TOF_TIME;   // Oneskorenie vypnutia vystrahy vystraznika po anulacii vystrahy
      ZH_ZD : TON_TIME;   // Oneskorenie medzi zdvihanim a spustanim zavor
   END_VAR
   VAR CONSTANT
      ZH_ZD_delay : Time := T#250ms;   // Cas pre oneskorenie medzi zdvihanim a spustanim zavor
   END_VAR
   VAR_TEMP   // added for the SCL form of the ladder/FBD networks
      _w1 : Bool;
      _w2 : Bool;
   END_VAR
BEGIN

REGION Network 1: Vyhodnotenie smeru jazdy KV
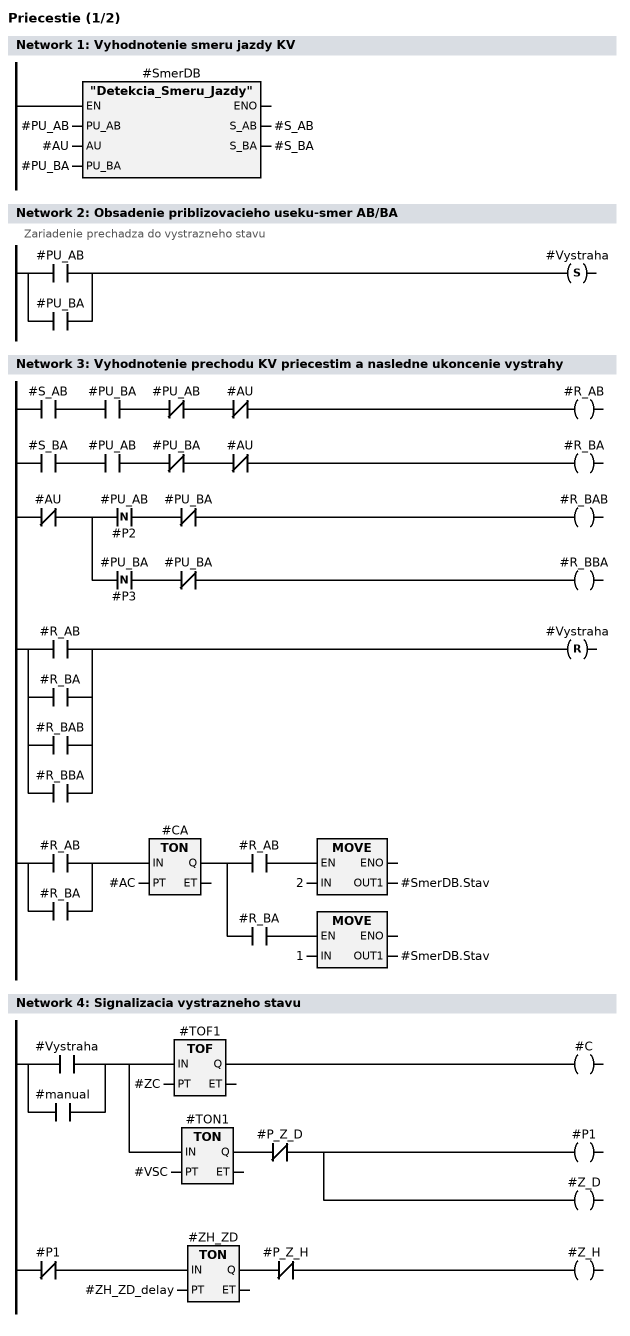
   RUNG wire#powerrail
      #SmerDB(PU_AB := #PU_AB, AU := #AU, PU_BA := #PU_BA, S_AB => #S_AB, S_BA => #S_BA)
   END_RUNG
   // the same network as SCL:
   #SmerDB(PU_AB := #PU_AB, AU := #AU, PU_BA := #PU_BA, S_AB => #S_AB, S_BA => #S_BA);   // "Detekcia_Smeru_Jazdy"
END_REGION

REGION Network 2: Obsadenie priblizovacieho useku-smer AB/BA
   // Zariadenie prechadza do vystrazneho stavu
   RUNG wire#powerrail
      Contact( #PU_AB )
      wire#w1
      S_Coil( #Vystraha )
   END_RUNG
   RUNG wire#powerrail
      Contact( #PU_BA )
   END_RUNG wire#w1
   // the same network as SCL:
   IF #PU_AB OR #PU_BA THEN #Vystraha := TRUE; END_IF;
END_REGION

REGION Network 3: Vyhodnotenie prechodu KV priecestim a nasledne ukoncenie vystrahy
   #R_AB := #S_AB AND #PU_BA AND NOT #PU_AB AND NOT #AU;
   #R_BA := #S_BA AND #PU_AB AND NOT #PU_BA AND NOT #AU;
   #_w1 := NOT #AU AND NOT #PU_AB AND #P2;   // falling edge of #PU_AB
   #P2 := #PU_AB;
   #R_BAB := #_w1 AND NOT #PU_BA;
   #_w2 := NOT #AU AND NOT #PU_BA AND #P3;   // falling edge of #PU_BA
   #P3 := #PU_BA;
   #R_BBA := #_w2 AND NOT #PU_BA;
   IF #R_AB OR #R_BA OR #R_BAB OR #R_BBA THEN #Vystraha := FALSE; END_IF;
   #CA(IN := #R_AB OR #R_BA, PT := #AC);   // TON
   IF #CA.Q AND #R_AB THEN #SmerDB.Stav := 2; END_IF;
   IF #CA.Q AND #R_BA THEN #SmerDB.Stav := 1; END_IF;
END_REGION

REGION Network 4: Signalizacia vystrazneho stavu
   #_w1 := #Vystraha OR #manual;
   #TOF1(IN := #_w1, PT := #ZC);   // TOF
   #C := #TOF1.Q;
   #TON1(IN := #_w1, PT := #VSC);   // TON
   #P1 := #TON1.Q AND NOT #P_Z_D;
   #Z_D := #P1;
   #ZH_ZD(IN := NOT #P1, PT := #ZH_ZD_delay);   // TON
   #Z_H := #ZH_ZD.Q AND NOT #P_Z_H;
END_REGION

REGION Network 5: Signalizacia zakladneho stavu
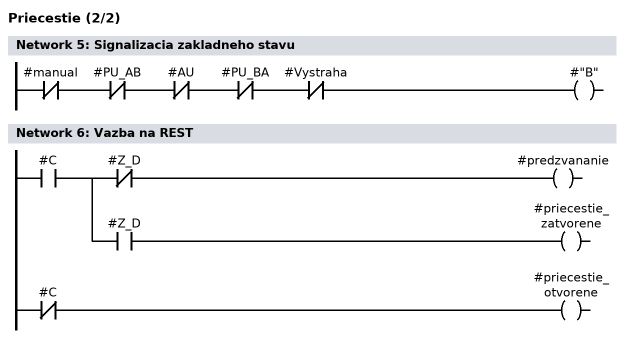
   RUNG wire#powerrail
      I_Contact( #manual )
      I_Contact( #PU_AB )
      I_Contact( #AU )
      I_Contact( #PU_BA )
      I_Contact( #Vystraha )
      Coil( #"B" )
   END_RUNG
   // the same network as SCL:
   #"B" := NOT #manual AND NOT #PU_AB AND NOT #AU AND NOT #PU_BA AND NOT #Vystraha;
END_REGION

REGION Network 6: Vazba na REST
   RUNG wire#powerrail
      Contact( #C )
      wire#w1
      I_Contact( #Z_D )
      Coil( #predzvananie )
   END_RUNG
   RUNG wire#w1
      Contact( #Z_D )
      Coil( #priecestie_zatvorene )
   END_RUNG
   RUNG wire#powerrail
      I_Contact( #C )
      Coil( #priecestie_otvorene )
   END_RUNG
   // the same network as SCL:
   #predzvananie := #C AND NOT #Z_D;
   #priecestie_zatvorene := #C AND #Z_D;
   #priecestie_otvorene := NOT #C;
END_REGION
END_FUNCTION_BLOCK

FUNCTION_BLOCK "Autoblok"   // FB3, LAD
{ S7_Optimized_Access := 'TRUE' }
VERSION : 0.1
   VAR_INPUT
      usek_za_nav : Bool;
      stav_nasl_nav : Byte;
      bikac : Bool;
      Trat_suhlas : Bool;
      smer_Nav : Bool;   // 0-lichy, 1-sudy
   END_VAR
   VAR_OUTPUT
      zlta : Bool;
      zelena : Bool;
      cervena : Bool;
   END_VAR
   VAR
      stav : Byte;   // 0-volno, 1-vystraha, 2-stoj, 3-ocakavaj_40, 4-40_a_vystraha
   END_VAR
   VAR_TEMP   // added for the SCL form of the ladder/FBD networks
      _w1 : Bool;
      _w2 : Bool;
      _w3 : Bool;
      _w4 : Bool;
   END_VAR
BEGIN

REGION Network 1
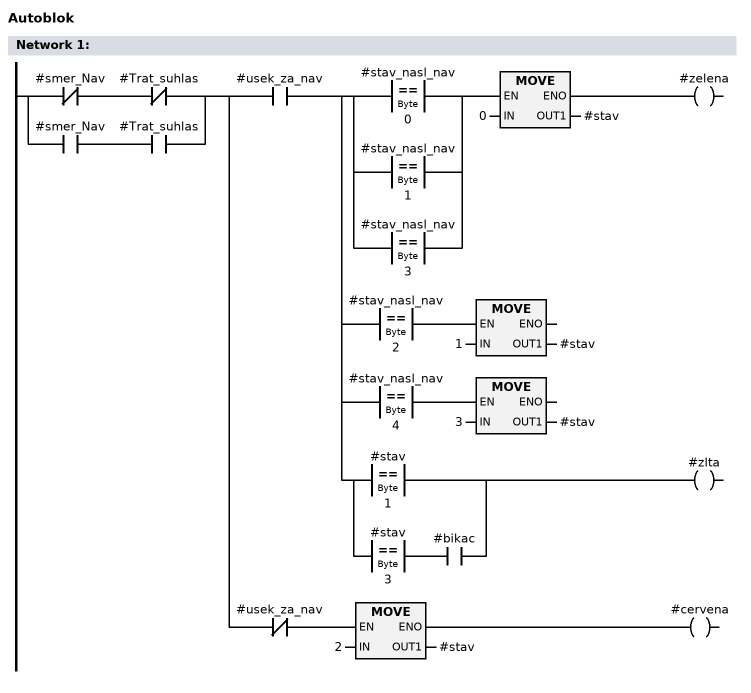
   RUNG wire#powerrail
      I_Contact( #smer_Nav )
      I_Contact( #Trat_suhlas )
      wire#w1
      Contact( #usek_za_nav )
      wire#w2
      { S7_Templates := "SrcType := Byte" } EQ_Contact(in1 := #stav_nasl_nav, in2 := 0)
      wire#w3
      Move(in := 0, out1 => #stav)
      Coil( #zelena )
   END_RUNG
   RUNG wire#powerrail
      Contact( #smer_Nav )
      Contact( #Trat_suhlas )
   END_RUNG wire#w1
   RUNG wire#w2
      { S7_Templates := "SrcType := Byte" } EQ_Contact(in1 := #stav_nasl_nav, in2 := 1)
   END_RUNG wire#w3
   RUNG wire#w2
      { S7_Templates := "SrcType := Byte" } EQ_Contact(in1 := #stav_nasl_nav, in2 := 3)
   END_RUNG wire#w3
   RUNG wire#w2
      { S7_Templates := "SrcType := Byte" } EQ_Contact(in1 := #stav_nasl_nav, in2 := 2)
      Move(in := 1, out1 => #stav)
   END_RUNG
   RUNG wire#w2
      { S7_Templates := "SrcType := Byte" } EQ_Contact(in1 := #stav_nasl_nav, in2 := 4)
      Move(in := 3, out1 => #stav)
   END_RUNG
   RUNG wire#w2
      { S7_Templates := "SrcType := Byte" } EQ_Contact(in1 := #stav, in2 := 1)
      wire#w4
      Coil( #zlta )
   END_RUNG
   RUNG wire#w2
      { S7_Templates := "SrcType := Byte" } EQ_Contact(in1 := #stav, in2 := 3)
      Contact( #bikac )
   END_RUNG wire#w4
   RUNG wire#w1
      I_Contact( #usek_za_nav )
      Move(in := 2, out1 => #stav)
      Coil( #cervena )
   END_RUNG
   // the same network as SCL:
   #_w1 := (NOT #smer_Nav AND NOT #Trat_suhlas) OR (#smer_Nav AND #Trat_suhlas);
   #_w2 := #_w1 AND #usek_za_nav;
   #_w3 := #_w2 AND ((#stav_nasl_nav = 0) OR (#stav_nasl_nav = 1) OR (#stav_nasl_nav = 3));
   IF #_w3 THEN #stav := 0; END_IF;
   #zelena := #_w3;
   IF #_w2 AND (#stav_nasl_nav = 2) THEN #stav := 1; END_IF;
   IF #_w2 AND (#stav_nasl_nav = 4) THEN #stav := 3; END_IF;
   #zlta := #_w2 AND ((#stav = 1) OR ((#stav = 3) AND #bikac));
   #_w4 := #_w1 AND NOT #usek_za_nav;
   IF #_w4 THEN #stav := 2; END_IF;
   #cervena := #_w4;
END_REGION
END_FUNCTION_BLOCK

FUNCTION_BLOCK "Radosina"   // FB4, LAD
{ S7_Optimized_Access := 'TRUE' }
VERSION : 0.1
   VAR_INPUT
      smer_v1 : Bool;   // 1->plus, 0->minus
      stav_AB19 : Int;   // 0->stoj, 1->vystraha, 2->volno, 4->zhasnute
      "medzist_usek_RAD-ZBE" : Bool;
      stavL1 : Byte;   // 0->stoj, 1->volno, 2->posun, 3->PN
      stavL2 : Byte;   // 0->stoj, 1->volno, 2->posun, 3->PN
      stavS : Byte;   // 0->stoj, 1->volno, 3->PN
      stavSe1 : Byte;   // 0->stoj, 2->posun
      prerusovac : Bool;
   END_VAR
   VAR_OUTPUT
      L1_zl : Bool;
      L1_ze : Bool;
      L1_ce : Bool;
      L1_bi : Bool;
      L2_zl_h : Bool;
      L2_ze : Bool;
      L2_ce : Bool;
      L2_bi : Bool;
      L2_zl_d : Bool;
      S_zl_h : Bool;
      S_ce : Bool;
      S_bi : Bool;
      S_zl_d : Bool;
      Se1_bi : Bool;
      Se1_mo : Bool;
      volnost_mu : Bool;   // volnost medzist. useku
   END_VAR
   VAR
      stavNavS : Byte;   // 0-volno, 1-vystraha, 2-stoj, 3-ocakavaj_40, 4-40_a_vystraha
   END_VAR
   VAR_TEMP   // added for the SCL form of the ladder/FBD networks
      _w1 : Bool;
      _w2 : Bool;
   END_VAR
BEGIN

REGION Network 1: volnost medzist. useku
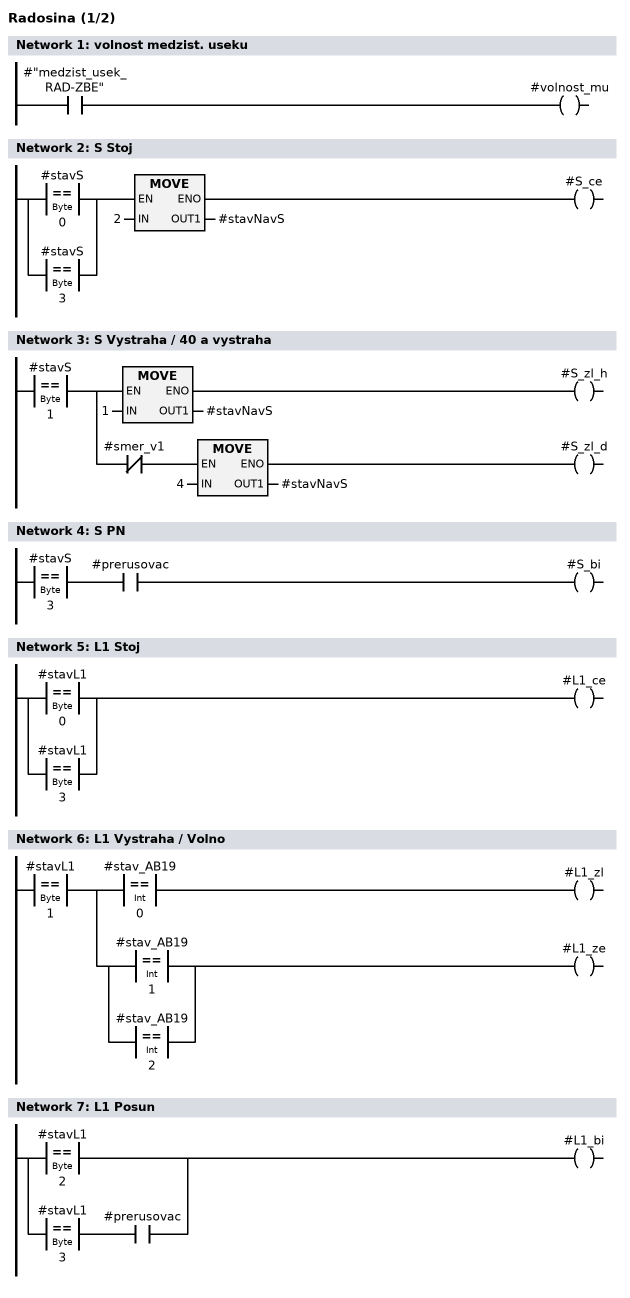
   RUNG wire#powerrail
      Contact( #"medzist_usek_RAD-ZBE" )
      Coil( #volnost_mu )
   END_RUNG
   // the same network as SCL:
   #volnost_mu := #"medzist_usek_RAD-ZBE";
END_REGION

REGION Network 2: S Stoj
   RUNG wire#powerrail
      { S7_Templates := "SrcType := Byte" } EQ_Contact(in1 := #stavS, in2 := 0)
      wire#w1
      Move(in := 2, out1 => #stavNavS)
      Coil( #S_ce )
   END_RUNG
   RUNG wire#powerrail
      { S7_Templates := "SrcType := Byte" } EQ_Contact(in1 := #stavS, in2 := 3)
   END_RUNG wire#w1
   // the same network as SCL:
   #_w1 := (#stavS = 0) OR (#stavS = 3);
   IF #_w1 THEN #stavNavS := 2; END_IF;
   #S_ce := #_w1;
END_REGION

REGION Network 3: S Vystraha / 40 a vystraha
   RUNG wire#powerrail
      { S7_Templates := "SrcType := Byte" } EQ_Contact(in1 := #stavS, in2 := 1)
      wire#w1
      Move(in := 1, out1 => #stavNavS)
      Coil( #S_zl_h )
   END_RUNG
   RUNG wire#w1
      I_Contact( #smer_v1 )
      Move(in := 4, out1 => #stavNavS)
      Coil( #S_zl_d )
   END_RUNG
   // the same network as SCL:
   #_w1 := #stavS = 1;
   IF #_w1 THEN #stavNavS := 1; END_IF;
   #S_zl_h := #_w1;
   #_w2 := #_w1 AND NOT #smer_v1;
   IF #_w2 THEN #stavNavS := 4; END_IF;
   #S_zl_d := #_w2;
END_REGION

REGION Network 4: S PN
   RUNG wire#powerrail
      { S7_Templates := "SrcType := Byte" } EQ_Contact(in1 := #stavS, in2 := 3)
      Contact( #prerusovac )
      Coil( #S_bi )
   END_RUNG
   // the same network as SCL:
   #S_bi := (#stavS = 3) AND #prerusovac;
END_REGION

REGION Network 5: L1 Stoj
   RUNG wire#powerrail
      { S7_Templates := "SrcType := Byte" } EQ_Contact(in1 := #stavL1, in2 := 0)
      wire#w1
      Coil( #L1_ce )
   END_RUNG
   RUNG wire#powerrail
      { S7_Templates := "SrcType := Byte" } EQ_Contact(in1 := #stavL1, in2 := 3)
   END_RUNG wire#w1
   // the same network as SCL:
   #L1_ce := (#stavL1 = 0) OR (#stavL1 = 3);
END_REGION

REGION Network 6: L1 Vystraha / Volno
   RUNG wire#powerrail
      { S7_Templates := "SrcType := Byte" } EQ_Contact(in1 := #stavL1, in2 := 1)
      wire#w1
      { S7_Templates := "SrcType := Int" } EQ_Contact(in1 := #stav_AB19, in2 := 0)
      Coil( #L1_zl )
   END_RUNG
   RUNG wire#w1
      { S7_Templates := "SrcType := Int" } EQ_Contact(in1 := #stav_AB19, in2 := 1)
      wire#w2
      Coil( #L1_ze )
   END_RUNG
   RUNG wire#w1
      { S7_Templates := "SrcType := Int" } EQ_Contact(in1 := #stav_AB19, in2 := 2)
   END_RUNG wire#w2
   // the same network as SCL:
   #_w1 := #stavL1 = 1;
   #L1_zl := #_w1 AND (#stav_AB19 = 0);
   #L1_ze := #_w1 AND ((#stav_AB19 = 1) OR (#stav_AB19 = 2));
END_REGION

REGION Network 7: L1 Posun
   RUNG wire#powerrail
      { S7_Templates := "SrcType := Byte" } EQ_Contact(in1 := #stavL1, in2 := 2)
      wire#w1
      Coil( #L1_bi )
   END_RUNG
   RUNG wire#powerrail
      { S7_Templates := "SrcType := Byte" } EQ_Contact(in1 := #stavL1, in2 := 3)
      Contact( #prerusovac )
   END_RUNG wire#w1
   // the same network as SCL:
   #L1_bi := (#stavL1 = 2) OR ((#stavL1 = 3) AND #prerusovac);
END_REGION

REGION Network 8: L2 Stoj
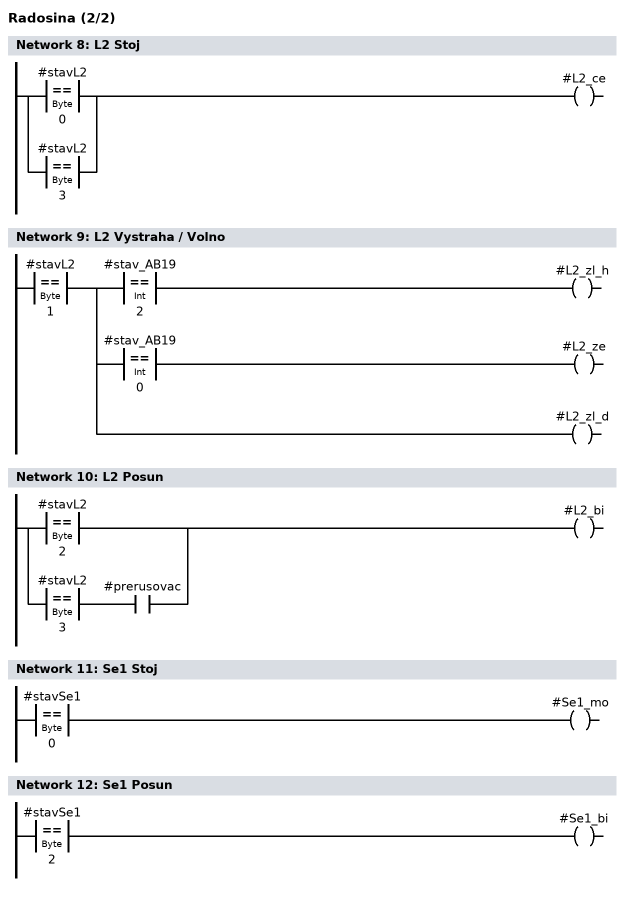
   RUNG wire#powerrail
      { S7_Templates := "SrcType := Byte" } EQ_Contact(in1 := #stavL2, in2 := 0)
      wire#w1
      Coil( #L2_ce )
   END_RUNG
   RUNG wire#powerrail
      { S7_Templates := "SrcType := Byte" } EQ_Contact(in1 := #stavL2, in2 := 3)
   END_RUNG wire#w1
   // the same network as SCL:
   #L2_ce := (#stavL2 = 0) OR (#stavL2 = 3);
END_REGION

REGION Network 9: L2 Vystraha / Volno
   RUNG wire#powerrail
      { S7_Templates := "SrcType := Byte" } EQ_Contact(in1 := #stavL2, in2 := 1)
      wire#w1
      { S7_Templates := "SrcType := Int" } EQ_Contact(in1 := #stav_AB19, in2 := 2)
      Coil( #L2_zl_h )
   END_RUNG
   RUNG wire#w1
      { S7_Templates := "SrcType := Int" } EQ_Contact(in1 := #stav_AB19, in2 := 0)
      Coil( #L2_ze )
   END_RUNG
   RUNG wire#w1
      Coil( #L2_zl_d )
   END_RUNG
   // the same network as SCL:
   #_w1 := #stavL2 = 1;
   #L2_zl_h := #_w1 AND (#stav_AB19 = 2);
   #L2_ze := #_w1 AND (#stav_AB19 = 0);
   #L2_zl_d := #_w1;
END_REGION

REGION Network 10: L2 Posun
   RUNG wire#powerrail
      { S7_Templates := "SrcType := Byte" } EQ_Contact(in1 := #stavL2, in2 := 2)
      wire#w1
      Coil( #L2_bi )
   END_RUNG
   RUNG wire#powerrail
      { S7_Templates := "SrcType := Byte" } EQ_Contact(in1 := #stavL2, in2 := 3)
      Contact( #prerusovac )
   END_RUNG wire#w1
   // the same network as SCL:
   #L2_bi := (#stavL2 = 2) OR ((#stavL2 = 3) AND #prerusovac);
END_REGION

REGION Network 11: Se1 Stoj
   RUNG wire#powerrail
      { S7_Templates := "SrcType := Byte" } EQ_Contact(in1 := #stavSe1, in2 := 0)
      Coil( #Se1_mo )
   END_RUNG
   // the same network as SCL:
   #Se1_mo := #stavSe1 = 0;
END_REGION

REGION Network 12: Se1 Posun
   RUNG wire#powerrail
      { S7_Templates := "SrcType := Byte" } EQ_Contact(in1 := #stavSe1, in2 := 2)
      Coil( #Se1_bi )
   END_RUNG
   // the same network as SCL:
   #Se1_bi := #stavSe1 = 2;
END_REGION
END_FUNCTION_BLOCK

FUNCTION_BLOCK "Zbehy"   // FB5, LAD
{ S7_Optimized_Access := 'TRUE' }
VERSION : 0.1
   VAR_INPUT
      "smer_v1-v2" : Bool;   // 1->plus, 0->minus
      smer_v3 : Bool;   // 1->plus, 0->minus
      stav_AB40 : Int;   // 0->stoj, 1->vystraha, 2->volno, 4->zhasnute
      "medzist_usek_RAD-ZBE" : Bool;
      "medzist_usek_ZBE-HLO" : Bool;
      TU_pred_S : Bool;
      TU_za_S : Bool;
      stavL : Byte;   // 0->stoj, 1->volno, 3->PN
      stavBL : Byte;   // 0->stoj, 1->volno, 3->PN
      stavL1 : Byte;   // 0->stoj, 1->volno, 2->posun, 3->PN
      stavL2 : Byte;   // 0->stoj, 1->volno, 2->posun, 3->PN
      stavS1 : Byte;   // 0->stoj, 1->volno, 2->posun, 3->PN
      stavS2 : Byte;   // 0->stoj, 1->volno, 2->posun, 3->PN
      stavS : Byte;   // 0->stoj, 1->volno, 3->PN
      stavSe1 : Byte;   // 0->stoj, 2->posun
      stavSe2 : Byte;   // 0->stoj, 2->posun
      stavSe3 : Byte;   // 0->stoj, 2->posun
      prerusovac : Bool;
      "OD_RAD-k1" : Bool;
      "OD_LUZ-k2" : Bool;
      "OD_HLO-k1" : Bool;
   END_VAR
   VAR_OUTPUT
      volnost_MU_HLO : Bool;
      S1_zl_h : Bool;
      S1_ze : Bool;
      S1_ce : Bool;
      S1_bi : Bool;
      S2_zl_h : Bool;
      S2_ze : Bool;
      S2_ce : Bool;
      S2_bi : Bool;
      S2_zl_d : Bool;
      L_zl_h : Bool;
      L_ze : Bool;
      L_ce : Bool;
      L_bi : Bool;
      L_zl_d : Bool;
      BL_zl_h : Bool;
      BL_ze : Bool;
      BL_ce : Bool;
      BL_bi : Bool;
      BL_zl_d : Bool;
      PrBL_ze : Bool;
      PrBL_zl : Bool;
      Se1_bi : Bool;
      Se1_mo : Bool;
      Se2_bi : Bool;
      Se2_mo : Bool;
      S_zl_h : Bool;
      S_ze : Bool;
      S_ce : Bool;
      S_bi : Bool;
      S_zl_d : Bool;
      PrS_ze : Bool;
      PrS_zl : Bool;
      L1_ze : Bool;
      L1_ce : Bool;
      L1_bi : Bool;
      L2_ze : Bool;
      L2_ce : Bool;
      L2_bi : Bool;
      L2_zl_d : Bool;
      Se3_mo : Bool;
      Se3_bi : Bool;
      odoslana_odhlaska : Bool := true;
   END_VAR
   VAR_IN_OUT
      dosla_predhlaska : Bool;
   END_VAR
   VAR
      stavNavL : Byte;   // 0-volno, 1-vystraha, 2-stoj, 3-ocakavaj_40, 4-40_a_vystraha
      vjazd : Bool;
   END_VAR
   VAR_TEMP   // added for the SCL form of the ladder/FBD networks
      _w1 : Bool;
   END_VAR
BEGIN

REGION Network 1: volnost medzist. useku
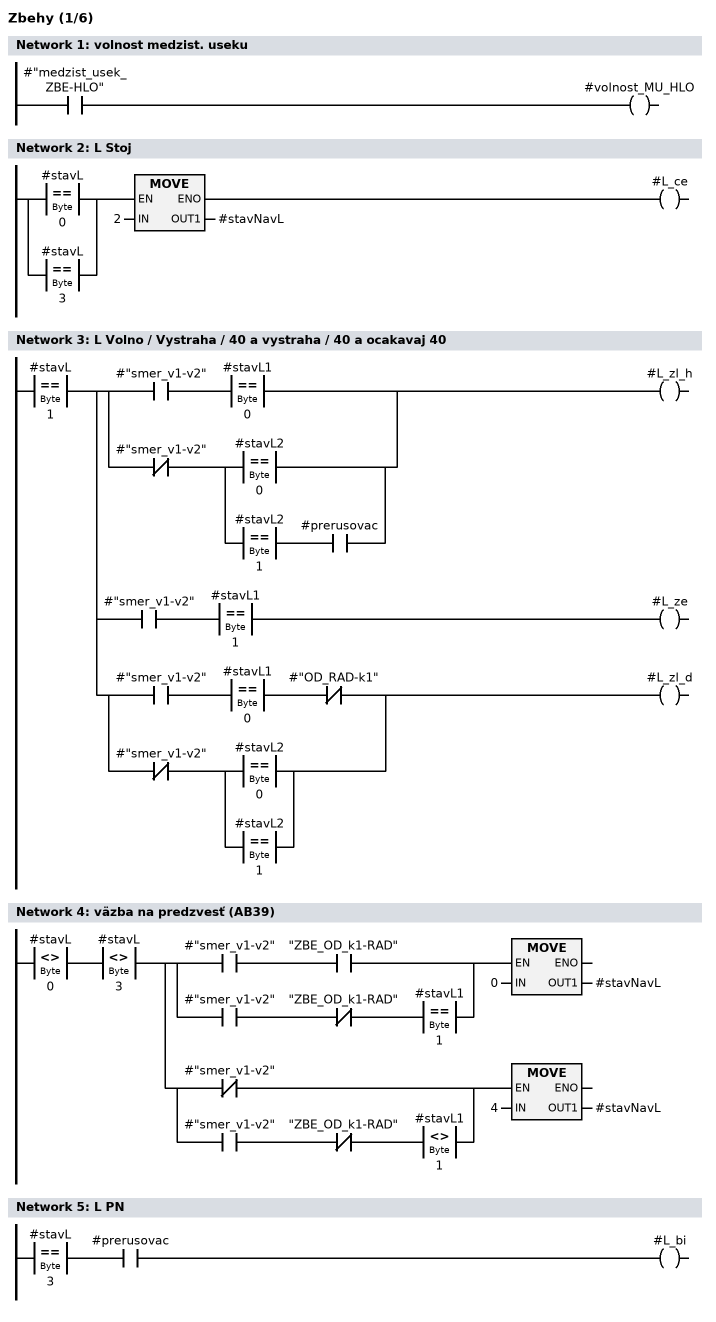
   RUNG wire#powerrail
      Contact( #"medzist_usek_ZBE-HLO" )
      Coil( #volnost_MU_HLO )
   END_RUNG
   // the same network as SCL:
   #volnost_MU_HLO := #"medzist_usek_ZBE-HLO";
END_REGION

REGION Network 2: L Stoj
   RUNG wire#powerrail
      { S7_Templates := "SrcType := Byte" } EQ_Contact(in1 := #stavL, in2 := 0)
      wire#w1
      Move(in := 2, out1 => #stavNavL)
      Coil( #L_ce )
   END_RUNG
   RUNG wire#powerrail
      { S7_Templates := "SrcType := Byte" } EQ_Contact(in1 := #stavL, in2 := 3)
   END_RUNG wire#w1
   // the same network as SCL:
   #_w1 := (#stavL = 0) OR (#stavL = 3);
   IF #_w1 THEN #stavNavL := 2; END_IF;
   #L_ce := #_w1;
END_REGION

REGION Network 3: L Volno / Vystraha / 40 a vystraha / 40 a ocakavaj 40
   RUNG wire#powerrail
      { S7_Templates := "SrcType := Byte" } EQ_Contact(in1 := #stavL, in2 := 1)
      wire#w1
      Contact( #"smer_v1-v2" )
      { S7_Templates := "SrcType := Byte" } EQ_Contact(in1 := #stavL1, in2 := 0)
      wire#w2
      Coil( #L_zl_h )
   END_RUNG
   RUNG wire#w1
      I_Contact( #"smer_v1-v2" )
      wire#w3
      { S7_Templates := "SrcType := Byte" } EQ_Contact(in1 := #stavL2, in2 := 0)
   END_RUNG wire#w2
   RUNG wire#w3
      { S7_Templates := "SrcType := Byte" } EQ_Contact(in1 := #stavL2, in2 := 1)
      Contact( #prerusovac )
   END_RUNG wire#w2
   RUNG wire#w1
      Contact( #"smer_v1-v2" )
      { S7_Templates := "SrcType := Byte" } EQ_Contact(in1 := #stavL1, in2 := 1)
      Coil( #L_ze )
   END_RUNG
   RUNG wire#w1
      Contact( #"smer_v1-v2" )
      { S7_Templates := "SrcType := Byte" } EQ_Contact(in1 := #stavL1, in2 := 0)
      I_Contact( #"OD_RAD-k1" )
      wire#w4
      Coil( #L_zl_d )
   END_RUNG
   RUNG wire#w1
      I_Contact( #"smer_v1-v2" )
      wire#w5
      { S7_Templates := "SrcType := Byte" } EQ_Contact(in1 := #stavL2, in2 := 0)
   END_RUNG wire#w4
   RUNG wire#w5
      { S7_Templates := "SrcType := Byte" } EQ_Contact(in1 := #stavL2, in2 := 1)
   END_RUNG wire#w4
   // the same network as SCL:
   #_w1 := #stavL = 1;
   #L_zl_h := #_w1 AND ((#"smer_v1-v2" AND (#stavL1 = 0)) OR (NOT #"smer_v1-v2" AND ((#stavL2 = 0) OR ((#stavL2 = 1) AND #prerusovac))));
   #L_ze := #_w1 AND #"smer_v1-v2" AND (#stavL1 = 1);
   #L_zl_d := #_w1 AND ((#"smer_v1-v2" AND (#stavL1 = 0) AND NOT #"OD_RAD-k1") OR (NOT #"smer_v1-v2" AND ((#stavL2 = 0) OR (#stavL2 = 1))));
END_REGION

REGION Network 4: väzba na predzvesť (AB39)
   RUNG wire#powerrail
      { S7_Templates := "SrcType := Byte" } NE_Contact(in1 := #stavL, in2 := 0)
      { S7_Templates := "SrcType := Byte" } NE_Contact(in1 := #stavL, in2 := 3)
      wire#w1
      Contact( #"smer_v1-v2" )
      Contact( "ZBE_OD_k1-RAD" )
      wire#w2
      Move(in := 0, out1 => #stavNavL)
   END_RUNG
   RUNG wire#w1
      Contact( #"smer_v1-v2" )
      I_Contact( "ZBE_OD_k1-RAD" )
      { S7_Templates := "SrcType := Byte" } EQ_Contact(in1 := #stavL1, in2 := 1)
   END_RUNG wire#w2
   RUNG wire#w1
      I_Contact( #"smer_v1-v2" )
      wire#w3
      Move(in := 4, out1 => #stavNavL)
   END_RUNG
   RUNG wire#w1
      Contact( #"smer_v1-v2" )
      I_Contact( "ZBE_OD_k1-RAD" )
      { S7_Templates := "SrcType := Byte" } NE_Contact(in1 := #stavL1, in2 := 1)
   END_RUNG wire#w3
   // the same network as SCL:
   #_w1 := (#stavL <> 0) AND (#stavL <> 3);
   IF #_w1 AND ((#"smer_v1-v2" AND "ZBE_OD_k1-RAD") OR (#"smer_v1-v2" AND NOT "ZBE_OD_k1-RAD" AND (#stavL1 = 1))) THEN
       #stavNavL := 0;
   END_IF;
   IF #_w1 AND (NOT #"smer_v1-v2" OR (#"smer_v1-v2" AND NOT "ZBE_OD_k1-RAD" AND (#stavL1 <> 1))) THEN
       #stavNavL := 4;
   END_IF;
END_REGION

REGION Network 5: L PN
   RUNG wire#powerrail
      { S7_Templates := "SrcType := Byte" } EQ_Contact(in1 := #stavL, in2 := 3)
      Contact( #prerusovac )
      Coil( #L_bi )
   END_RUNG
   // the same network as SCL:
   #L_bi := (#stavL = 3) AND #prerusovac;
END_REGION

REGION Network 6: BL Stoj
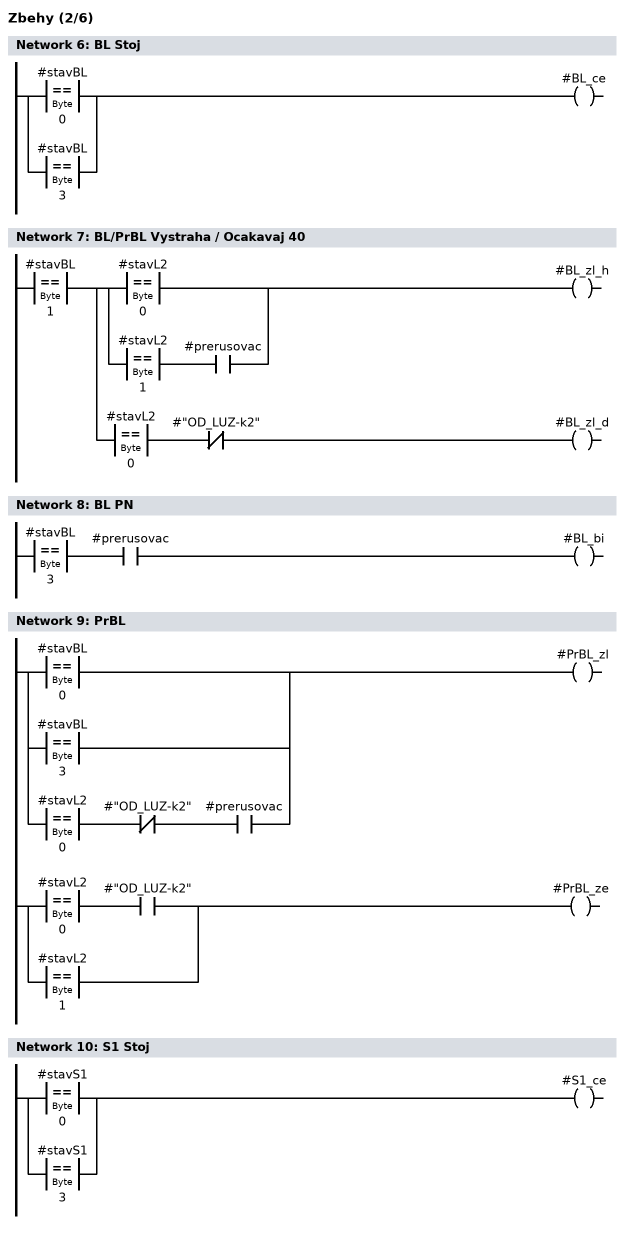
   RUNG wire#powerrail
      { S7_Templates := "SrcType := Byte" } EQ_Contact(in1 := #stavBL, in2 := 0)
      wire#w1
      Coil( #BL_ce )
   END_RUNG
   RUNG wire#powerrail
      { S7_Templates := "SrcType := Byte" } EQ_Contact(in1 := #stavBL, in2 := 3)
   END_RUNG wire#w1
   // the same network as SCL:
   #BL_ce := (#stavBL = 0) OR (#stavBL = 3);
END_REGION

REGION Network 7: BL/PrBL Vystraha / Ocakavaj 40
   RUNG wire#powerrail
      { S7_Templates := "SrcType := Byte" } EQ_Contact(in1 := #stavBL, in2 := 1)
      wire#w1
      { S7_Templates := "SrcType := Byte" } EQ_Contact(in1 := #stavL2, in2 := 0)
      wire#w2
      Coil( #BL_zl_h )
   END_RUNG
   RUNG wire#w1
      { S7_Templates := "SrcType := Byte" } EQ_Contact(in1 := #stavL2, in2 := 1)
      Contact( #prerusovac )
   END_RUNG wire#w2
   RUNG wire#w1
      { S7_Templates := "SrcType := Byte" } EQ_Contact(in1 := #stavL2, in2 := 0)
      I_Contact( #"OD_LUZ-k2" )
      Coil( #BL_zl_d )
   END_RUNG
   // the same network as SCL:
   #_w1 := #stavBL = 1;
   #BL_zl_h := #_w1 AND ((#stavL2 = 0) OR ((#stavL2 = 1) AND #prerusovac));
   #BL_zl_d := #_w1 AND (#stavL2 = 0) AND NOT #"OD_LUZ-k2";
END_REGION

REGION Network 8: BL PN
   RUNG wire#powerrail
      { S7_Templates := "SrcType := Byte" } EQ_Contact(in1 := #stavBL, in2 := 3)
      Contact( #prerusovac )
      Coil( #BL_bi )
   END_RUNG
   // the same network as SCL:
   #BL_bi := (#stavBL = 3) AND #prerusovac;
END_REGION

REGION Network 9: PrBL
   RUNG wire#powerrail
      { S7_Templates := "SrcType := Byte" } EQ_Contact(in1 := #stavBL, in2 := 0)
      wire#w1
      Coil( #PrBL_zl )
   END_RUNG
   RUNG wire#powerrail
      { S7_Templates := "SrcType := Byte" } EQ_Contact(in1 := #stavBL, in2 := 3)
   END_RUNG wire#w1
   RUNG wire#powerrail
      { S7_Templates := "SrcType := Byte" } EQ_Contact(in1 := #stavL2, in2 := 0)
      I_Contact( #"OD_LUZ-k2" )
      Contact( #prerusovac )
   END_RUNG wire#w1
   RUNG wire#powerrail
      { S7_Templates := "SrcType := Byte" } EQ_Contact(in1 := #stavL2, in2 := 0)
      Contact( #"OD_LUZ-k2" )
      wire#w2
      Coil( #PrBL_ze )
   END_RUNG
   RUNG wire#powerrail
      { S7_Templates := "SrcType := Byte" } EQ_Contact(in1 := #stavL2, in2 := 1)
   END_RUNG wire#w2
   // the same network as SCL:
   #PrBL_zl := (#stavBL = 0) OR (#stavBL = 3) OR ((#stavL2 = 0) AND NOT #"OD_LUZ-k2" AND #prerusovac);
   #PrBL_ze := ((#stavL2 = 0) AND #"OD_LUZ-k2") OR (#stavL2 = 1);
END_REGION

REGION Network 10: S1 Stoj
   RUNG wire#powerrail
      { S7_Templates := "SrcType := Byte" } EQ_Contact(in1 := #stavS1, in2 := 0)
      wire#w1
      Coil( #S1_ce )
   END_RUNG
   RUNG wire#powerrail
      { S7_Templates := "SrcType := Byte" } EQ_Contact(in1 := #stavS1, in2 := 3)
   END_RUNG wire#w1
   // the same network as SCL:
   #S1_ce := (#stavS1 = 0) OR (#stavS1 = 3);
END_REGION

REGION Network 11: S1 Vystraha / Volno
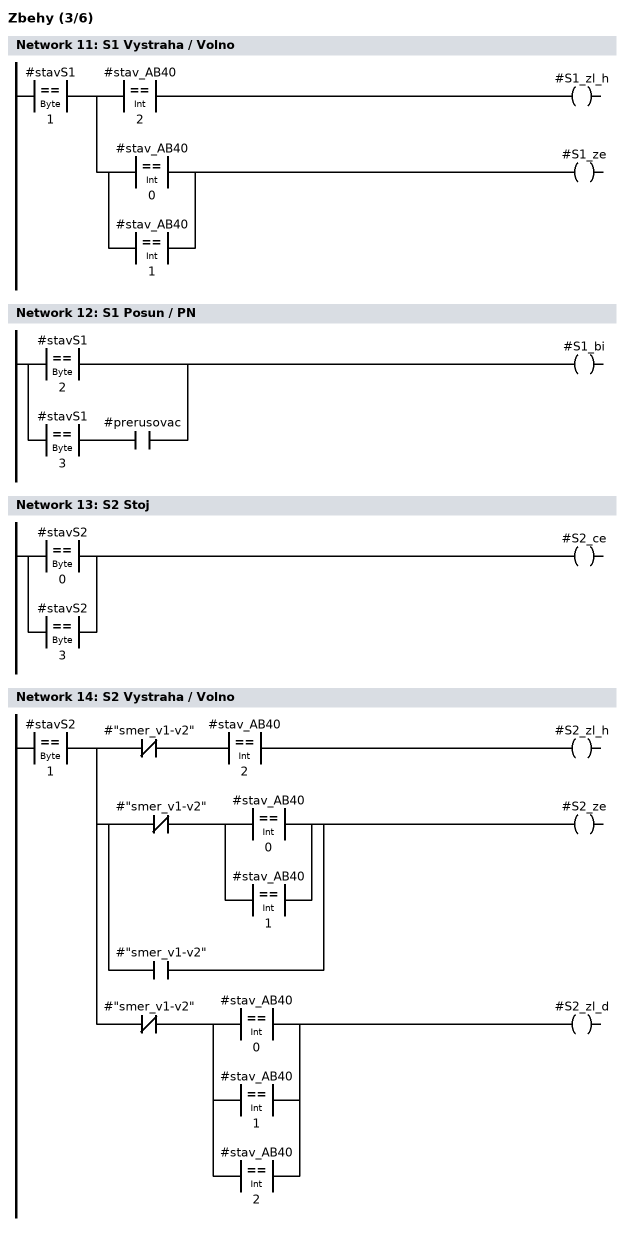
   RUNG wire#powerrail
      { S7_Templates := "SrcType := Byte" } EQ_Contact(in1 := #stavS1, in2 := 1)
      wire#w1
      { S7_Templates := "SrcType := Int" } EQ_Contact(in1 := #stav_AB40, in2 := 2)
      Coil( #S1_zl_h )
   END_RUNG
   RUNG wire#w1
      { S7_Templates := "SrcType := Int" } EQ_Contact(in1 := #stav_AB40, in2 := 0)
      wire#w2
      Coil( #S1_ze )
   END_RUNG
   RUNG wire#w1
      { S7_Templates := "SrcType := Int" } EQ_Contact(in1 := #stav_AB40, in2 := 1)
   END_RUNG wire#w2
   // the same network as SCL:
   #_w1 := #stavS1 = 1;
   #S1_zl_h := #_w1 AND (#stav_AB40 = 2);
   #S1_ze := #_w1 AND ((#stav_AB40 = 0) OR (#stav_AB40 = 1));
END_REGION

REGION Network 12: S1 Posun / PN
   RUNG wire#powerrail
      { S7_Templates := "SrcType := Byte" } EQ_Contact(in1 := #stavS1, in2 := 2)
      wire#w1
      Coil( #S1_bi )
   END_RUNG
   RUNG wire#powerrail
      { S7_Templates := "SrcType := Byte" } EQ_Contact(in1 := #stavS1, in2 := 3)
      Contact( #prerusovac )
   END_RUNG wire#w1
   // the same network as SCL:
   #S1_bi := (#stavS1 = 2) OR ((#stavS1 = 3) AND #prerusovac);
END_REGION

REGION Network 13: S2 Stoj
   RUNG wire#powerrail
      { S7_Templates := "SrcType := Byte" } EQ_Contact(in1 := #stavS2, in2 := 0)
      wire#w1
      Coil( #S2_ce )
   END_RUNG
   RUNG wire#powerrail
      { S7_Templates := "SrcType := Byte" } EQ_Contact(in1 := #stavS2, in2 := 3)
   END_RUNG wire#w1
   // the same network as SCL:
   #S2_ce := (#stavS2 = 0) OR (#stavS2 = 3);
END_REGION

REGION Network 14: S2 Vystraha / Volno
   RUNG wire#powerrail
      { S7_Templates := "SrcType := Byte" } EQ_Contact(in1 := #stavS2, in2 := 1)
      wire#w1
      I_Contact( #"smer_v1-v2" )
      { S7_Templates := "SrcType := Int" } EQ_Contact(in1 := #stav_AB40, in2 := 2)
      Coil( #S2_zl_h )
   END_RUNG
   RUNG wire#w1
      I_Contact( #"smer_v1-v2" )
      wire#w2
      { S7_Templates := "SrcType := Int" } EQ_Contact(in1 := #stav_AB40, in2 := 0)
      wire#w3
      Coil( #S2_ze )
   END_RUNG
   RUNG wire#w2
      { S7_Templates := "SrcType := Int" } EQ_Contact(in1 := #stav_AB40, in2 := 1)
   END_RUNG wire#w3
   RUNG wire#w1
      Contact( #"smer_v1-v2" )
   END_RUNG wire#w3
   RUNG wire#w1
      I_Contact( #"smer_v1-v2" )
      wire#w4
      { S7_Templates := "SrcType := Int" } EQ_Contact(in1 := #stav_AB40, in2 := 0)
      wire#w5
      Coil( #S2_zl_d )
   END_RUNG
   RUNG wire#w4
      { S7_Templates := "SrcType := Int" } EQ_Contact(in1 := #stav_AB40, in2 := 1)
   END_RUNG wire#w5
   RUNG wire#w4
      { S7_Templates := "SrcType := Int" } EQ_Contact(in1 := #stav_AB40, in2 := 2)
   END_RUNG wire#w5
   // the same network as SCL:
   #_w1 := #stavS2 = 1;
   #S2_zl_h := #_w1 AND NOT #"smer_v1-v2" AND (#stav_AB40 = 2);
   #S2_ze := #_w1 AND ((NOT #"smer_v1-v2" AND ((#stav_AB40 = 0) OR (#stav_AB40 = 1))) OR #"smer_v1-v2");
   #S2_zl_d := #_w1 AND NOT #"smer_v1-v2" AND ((#stav_AB40 = 0) OR (#stav_AB40 = 1) OR (#stav_AB40 = 2));
END_REGION

REGION Network 15: S2 Posun / PN
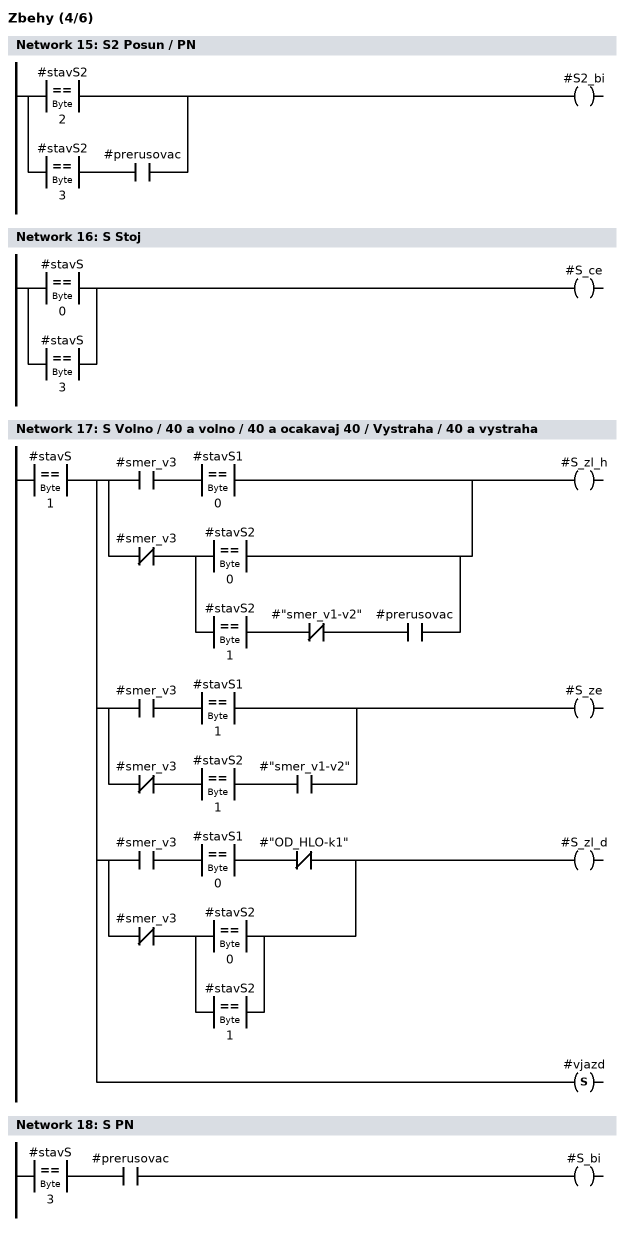
   RUNG wire#powerrail
      { S7_Templates := "SrcType := Byte" } EQ_Contact(in1 := #stavS2, in2 := 2)
      wire#w1
      Coil( #S2_bi )
   END_RUNG
   RUNG wire#powerrail
      { S7_Templates := "SrcType := Byte" } EQ_Contact(in1 := #stavS2, in2 := 3)
      Contact( #prerusovac )
   END_RUNG wire#w1
   // the same network as SCL:
   #S2_bi := (#stavS2 = 2) OR ((#stavS2 = 3) AND #prerusovac);
END_REGION

REGION Network 16: S Stoj
   RUNG wire#powerrail
      { S7_Templates := "SrcType := Byte" } EQ_Contact(in1 := #stavS, in2 := 0)
      wire#w1
      Coil( #S_ce )
   END_RUNG
   RUNG wire#powerrail
      { S7_Templates := "SrcType := Byte" } EQ_Contact(in1 := #stavS, in2 := 3)
   END_RUNG wire#w1
   // the same network as SCL:
   #S_ce := (#stavS = 0) OR (#stavS = 3);
END_REGION

REGION Network 17: S Volno / 40 a volno / 40 a ocakavaj 40 / Vystraha / 40 a vystraha
   RUNG wire#powerrail
      { S7_Templates := "SrcType := Byte" } EQ_Contact(in1 := #stavS, in2 := 1)
      wire#w1
      Contact( #smer_v3 )
      { S7_Templates := "SrcType := Byte" } EQ_Contact(in1 := #stavS1, in2 := 0)
      wire#w2
      Coil( #S_zl_h )
   END_RUNG
   RUNG wire#w1
      I_Contact( #smer_v3 )
      wire#w3
      { S7_Templates := "SrcType := Byte" } EQ_Contact(in1 := #stavS2, in2 := 0)
   END_RUNG wire#w2
   RUNG wire#w3
      { S7_Templates := "SrcType := Byte" } EQ_Contact(in1 := #stavS2, in2 := 1)
      I_Contact( #"smer_v1-v2" )
      Contact( #prerusovac )
   END_RUNG wire#w2
   RUNG wire#w1
      Contact( #smer_v3 )
      { S7_Templates := "SrcType := Byte" } EQ_Contact(in1 := #stavS1, in2 := 1)
      wire#w4
      Coil( #S_ze )
   END_RUNG
   RUNG wire#w1
      I_Contact( #smer_v3 )
      { S7_Templates := "SrcType := Byte" } EQ_Contact(in1 := #stavS2, in2 := 1)
      Contact( #"smer_v1-v2" )
   END_RUNG wire#w4
   RUNG wire#w1
      Contact( #smer_v3 )
      { S7_Templates := "SrcType := Byte" } EQ_Contact(in1 := #stavS1, in2 := 0)
      I_Contact( #"OD_HLO-k1" )
      wire#w5
      Coil( #S_zl_d )
   END_RUNG
   RUNG wire#w1
      I_Contact( #smer_v3 )
      wire#w6
      { S7_Templates := "SrcType := Byte" } EQ_Contact(in1 := #stavS2, in2 := 0)
   END_RUNG wire#w5
   RUNG wire#w6
      { S7_Templates := "SrcType := Byte" } EQ_Contact(in1 := #stavS2, in2 := 1)
   END_RUNG wire#w5
   RUNG wire#w1
      S_Coil( #vjazd )
   END_RUNG
   // the same network as SCL:
   #_w1 := #stavS = 1;
   #S_zl_h := #_w1 AND ((#smer_v3 AND (#stavS1 = 0)) OR (NOT #smer_v3 AND ((#stavS2 = 0) OR ((#stavS2 = 1) AND NOT #"smer_v1-v2" AND #prerusovac))));
   #S_ze := #_w1 AND ((#smer_v3 AND (#stavS1 = 1)) OR (NOT #smer_v3 AND (#stavS2 = 1) AND #"smer_v1-v2"));
   #S_zl_d := #_w1 AND ((#smer_v3 AND (#stavS1 = 0) AND NOT #"OD_HLO-k1") OR (NOT #smer_v3 AND ((#stavS2 = 0) OR (#stavS2 = 1))));
   IF #_w1 THEN #vjazd := TRUE; END_IF;
END_REGION

REGION Network 18: S PN
   RUNG wire#powerrail
      { S7_Templates := "SrcType := Byte" } EQ_Contact(in1 := #stavS, in2 := 3)
      Contact( #prerusovac )
      Coil( #S_bi )
   END_RUNG
   // the same network as SCL:
   #S_bi := (#stavS = 3) AND #prerusovac;
END_REGION

REGION Network 19: PrS
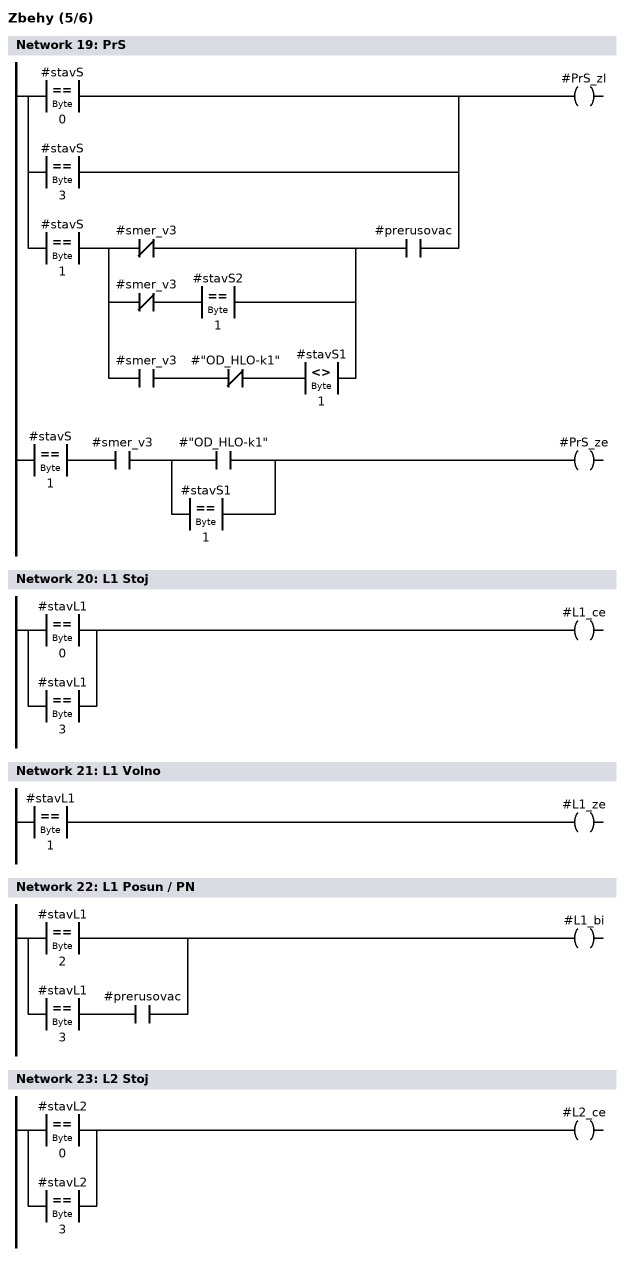
   RUNG wire#powerrail
      { S7_Templates := "SrcType := Byte" } EQ_Contact(in1 := #stavS, in2 := 0)
      wire#w1
      Coil( #PrS_zl )
   END_RUNG
   RUNG wire#powerrail
      { S7_Templates := "SrcType := Byte" } EQ_Contact(in1 := #stavS, in2 := 3)
   END_RUNG wire#w1
   RUNG wire#powerrail
      { S7_Templates := "SrcType := Byte" } EQ_Contact(in1 := #stavS, in2 := 1)
      wire#w2
      I_Contact( #smer_v3 )
      wire#w3
      Contact( #prerusovac )
   END_RUNG wire#w1
   RUNG wire#w2
      I_Contact( #smer_v3 )
      { S7_Templates := "SrcType := Byte" } EQ_Contact(in1 := #stavS2, in2 := 1)
   END_RUNG wire#w3
   RUNG wire#w2
      Contact( #smer_v3 )
      I_Contact( #"OD_HLO-k1" )
      { S7_Templates := "SrcType := Byte" } NE_Contact(in1 := #stavS1, in2 := 1)
   END_RUNG wire#w3
   RUNG wire#powerrail
      { S7_Templates := "SrcType := Byte" } EQ_Contact(in1 := #stavS, in2 := 1)
      Contact( #smer_v3 )
      wire#w4
      Contact( #"OD_HLO-k1" )
      wire#w5
      Coil( #PrS_ze )
   END_RUNG
   RUNG wire#w4
      { S7_Templates := "SrcType := Byte" } EQ_Contact(in1 := #stavS1, in2 := 1)
   END_RUNG wire#w5
   // the same network as SCL:
   #PrS_zl := (#stavS = 0) OR (#stavS = 3) OR ((#stavS = 1) AND (NOT #smer_v3 OR (NOT #smer_v3 AND (#stavS2 = 1)) OR (#smer_v3 AND NOT #"OD_HLO-k1" AND (#stavS1 <> 1))) AND #prerusovac);
   #PrS_ze := (#stavS = 1) AND #smer_v3 AND (#"OD_HLO-k1" OR (#stavS1 = 1));
END_REGION

REGION Network 20: L1 Stoj
   RUNG wire#powerrail
      { S7_Templates := "SrcType := Byte" } EQ_Contact(in1 := #stavL1, in2 := 0)
      wire#w1
      Coil( #L1_ce )
   END_RUNG
   RUNG wire#powerrail
      { S7_Templates := "SrcType := Byte" } EQ_Contact(in1 := #stavL1, in2 := 3)
   END_RUNG wire#w1
   // the same network as SCL:
   #L1_ce := (#stavL1 = 0) OR (#stavL1 = 3);
END_REGION

REGION Network 21: L1 Volno
   RUNG wire#powerrail
      { S7_Templates := "SrcType := Byte" } EQ_Contact(in1 := #stavL1, in2 := 1)
      Coil( #L1_ze )
   END_RUNG
   // the same network as SCL:
   #L1_ze := #stavL1 = 1;
END_REGION

REGION Network 22: L1 Posun / PN
   RUNG wire#powerrail
      { S7_Templates := "SrcType := Byte" } EQ_Contact(in1 := #stavL1, in2 := 2)
      wire#w1
      Coil( #L1_bi )
   END_RUNG
   RUNG wire#powerrail
      { S7_Templates := "SrcType := Byte" } EQ_Contact(in1 := #stavL1, in2 := 3)
      Contact( #prerusovac )
   END_RUNG wire#w1
   // the same network as SCL:
   #L1_bi := (#stavL1 = 2) OR ((#stavL1 = 3) AND #prerusovac);
END_REGION

REGION Network 23: L2 Stoj
   RUNG wire#powerrail
      { S7_Templates := "SrcType := Byte" } EQ_Contact(in1 := #stavL2, in2 := 0)
      wire#w1
      Coil( #L2_ce )
   END_RUNG
   RUNG wire#powerrail
      { S7_Templates := "SrcType := Byte" } EQ_Contact(in1 := #stavL2, in2 := 3)
   END_RUNG wire#w1
   // the same network as SCL:
   #L2_ce := (#stavL2 = 0) OR (#stavL2 = 3);
END_REGION

REGION Network 24: L2 Volno
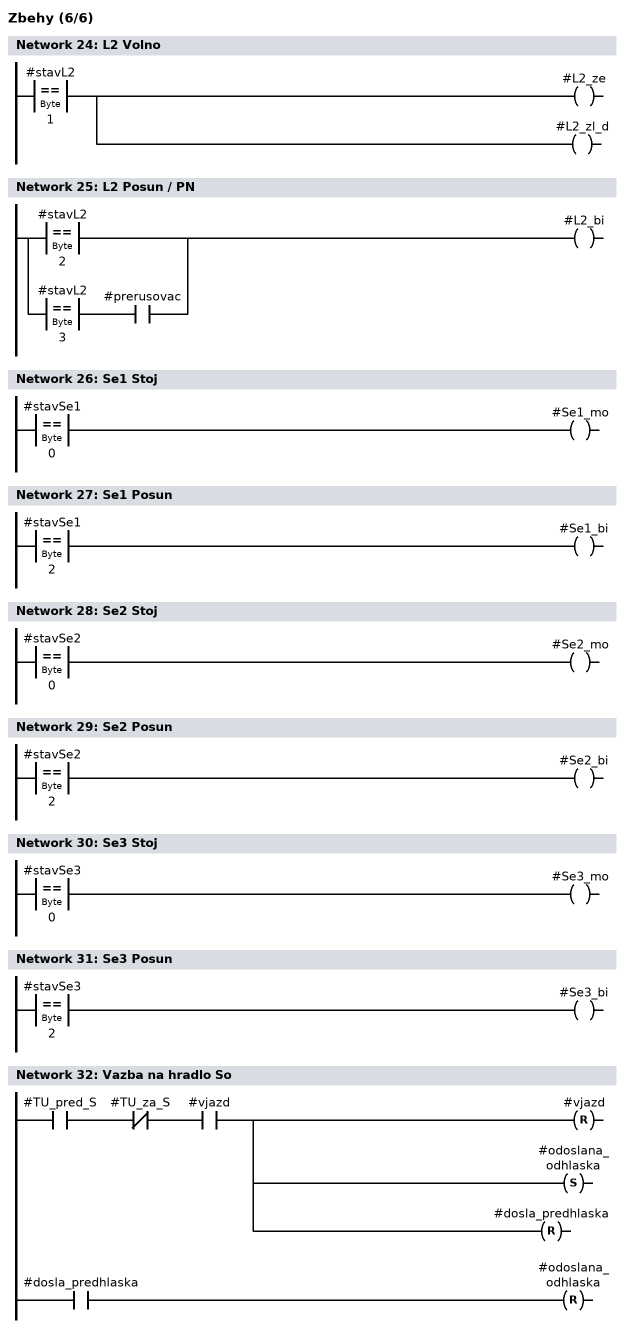
   RUNG wire#powerrail
      { S7_Templates := "SrcType := Byte" } EQ_Contact(in1 := #stavL2, in2 := 1)
      wire#w1
      Coil( #L2_ze )
   END_RUNG
   RUNG wire#w1
      Coil( #L2_zl_d )
   END_RUNG
   // the same network as SCL:
   #L2_ze := #stavL2 = 1;
   #L2_zl_d := #L2_ze;
END_REGION

REGION Network 25: L2 Posun / PN
   RUNG wire#powerrail
      { S7_Templates := "SrcType := Byte" } EQ_Contact(in1 := #stavL2, in2 := 2)
      wire#w1
      Coil( #L2_bi )
   END_RUNG
   RUNG wire#powerrail
      { S7_Templates := "SrcType := Byte" } EQ_Contact(in1 := #stavL2, in2 := 3)
      Contact( #prerusovac )
   END_RUNG wire#w1
   // the same network as SCL:
   #L2_bi := (#stavL2 = 2) OR ((#stavL2 = 3) AND #prerusovac);
END_REGION

REGION Network 26: Se1 Stoj
   RUNG wire#powerrail
      { S7_Templates := "SrcType := Byte" } EQ_Contact(in1 := #stavSe1, in2 := 0)
      Coil( #Se1_mo )
   END_RUNG
   // the same network as SCL:
   #Se1_mo := #stavSe1 = 0;
END_REGION

REGION Network 27: Se1 Posun
   RUNG wire#powerrail
      { S7_Templates := "SrcType := Byte" } EQ_Contact(in1 := #stavSe1, in2 := 2)
      Coil( #Se1_bi )
   END_RUNG
   // the same network as SCL:
   #Se1_bi := #stavSe1 = 2;
END_REGION

REGION Network 28: Se2 Stoj
   RUNG wire#powerrail
      { S7_Templates := "SrcType := Byte" } EQ_Contact(in1 := #stavSe2, in2 := 0)
      Coil( #Se2_mo )
   END_RUNG
   // the same network as SCL:
   #Se2_mo := #stavSe2 = 0;
END_REGION

REGION Network 29: Se2 Posun
   RUNG wire#powerrail
      { S7_Templates := "SrcType := Byte" } EQ_Contact(in1 := #stavSe2, in2 := 2)
      Coil( #Se2_bi )
   END_RUNG
   // the same network as SCL:
   #Se2_bi := #stavSe2 = 2;
END_REGION

REGION Network 30: Se3 Stoj
   RUNG wire#powerrail
      { S7_Templates := "SrcType := Byte" } EQ_Contact(in1 := #stavSe3, in2 := 0)
      Coil( #Se3_mo )
   END_RUNG
   // the same network as SCL:
   #Se3_mo := #stavSe3 = 0;
END_REGION

REGION Network 31: Se3 Posun
   RUNG wire#powerrail
      { S7_Templates := "SrcType := Byte" } EQ_Contact(in1 := #stavSe3, in2 := 2)
      Coil( #Se3_bi )
   END_RUNG
   // the same network as SCL:
   #Se3_bi := #stavSe3 = 2;
END_REGION

REGION Network 32: Vazba na hradlo So
   RUNG wire#powerrail
      Contact( #TU_pred_S )
      I_Contact( #TU_za_S )
      Contact( #vjazd )
      wire#w1
      R_Coil( #vjazd )
   END_RUNG
   RUNG wire#w1
      S_Coil( #odoslana_odhlaska )
   END_RUNG
   RUNG wire#w1
      R_Coil( #dosla_predhlaska )
   END_RUNG
   RUNG wire#powerrail
      Contact( #dosla_predhlaska )
      R_Coil( #odoslana_odhlaska )
   END_RUNG
   // the same network as SCL:
   #_w1 := #TU_pred_S AND NOT #TU_za_S AND #vjazd;
   IF #_w1 THEN
       #vjazd := FALSE;
       #odoslana_odhlaska := TRUE;
       #dosla_predhlaska := FALSE;
   END_IF;
   IF #dosla_predhlaska THEN #odoslana_odhlaska := FALSE; END_IF;
END_REGION
END_FUNCTION_BLOCK

FUNCTION_BLOCK "Hlohovec"   // FB6, LAD
{ S7_Optimized_Access := 'TRUE' }
VERSION : 0.1
   VAR_INPUT
      smer_v1 : Bool;   // 1->plus, 0->minus
      medzist_usek : Bool;
      TU_pred_L : Bool;
      TU_za_L : Bool;
      stavL : Byte;   // 0->stoj, 1->volno, 3->PN
      stavS1 : Byte;   // 0->stoj, 1->volno, 2->posun, 3->PN
      stavS2 : Byte;   // 0->stoj, 1->volno, 2->posun, 3->PN
      stavSe1 : Byte;   // 0->stoj, 2->posun
      prerusovac : Bool;
   END_VAR
   VAR_OUTPUT
      volnost_mu : Bool;   // volnost medzist. useku
      L_zl_h : Bool;
      L_ce : Bool;
      L_bi : Bool;
      L_zl_d : Bool;
      PrL_ze : Bool;
      PrL_zl : Bool;
      S1_ze : Bool;
      S1_ce : Bool;
      S1_bi : Bool;
      S2_ze : Bool;
      S2_ce : Bool;
      S2_bi : Bool;
      S2_zl_d : Bool;
      Se1_mo : Bool;
      Se1_bi : Bool;
      odoslana_odhlaska : Bool := true;
   END_VAR
   VAR_IN_OUT
      dosla_predhlaska : Bool;
   END_VAR
   VAR
      vjazd : Bool;
   END_VAR
   VAR_TEMP   // added for the SCL form of the ladder/FBD networks
      _w1 : Bool;
   END_VAR
BEGIN

REGION Network 1: volnost medzist. useku
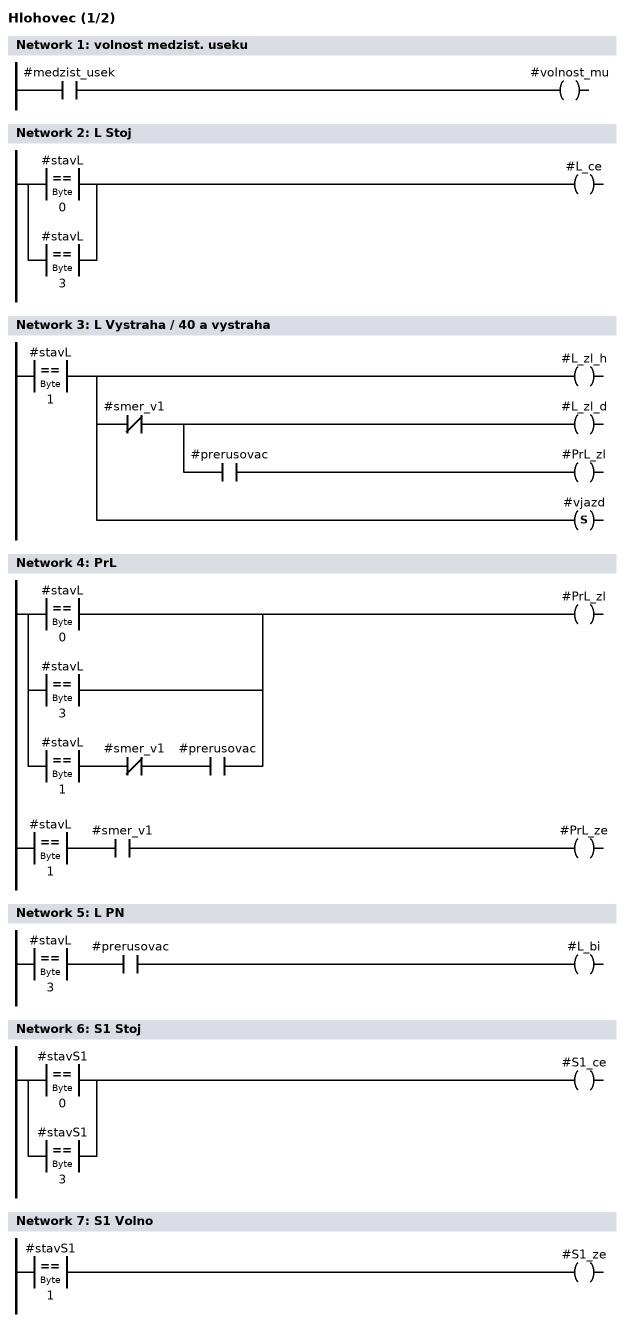
   RUNG wire#powerrail
      Contact( #medzist_usek )
      Coil( #volnost_mu )
   END_RUNG
   // the same network as SCL:
   #volnost_mu := #medzist_usek;
END_REGION

REGION Network 2: L Stoj
   RUNG wire#powerrail
      { S7_Templates := "SrcType := Byte" } EQ_Contact(in1 := #stavL, in2 := 0)
      wire#w1
      Coil( #L_ce )
   END_RUNG
   RUNG wire#powerrail
      { S7_Templates := "SrcType := Byte" } EQ_Contact(in1 := #stavL, in2 := 3)
   END_RUNG wire#w1
   // the same network as SCL:
   #L_ce := (#stavL = 0) OR (#stavL = 3);
END_REGION

REGION Network 3: L Vystraha / 40 a vystraha
   RUNG wire#powerrail
      { S7_Templates := "SrcType := Byte" } EQ_Contact(in1 := #stavL, in2 := 1)
      wire#w1
      Coil( #L_zl_h )
   END_RUNG
   RUNG wire#w1
      I_Contact( #smer_v1 )
      wire#w2
      Coil( #L_zl_d )
   END_RUNG
   RUNG wire#w2
      Contact( #prerusovac )
      Coil( #PrL_zl )
   END_RUNG
   RUNG wire#w1
      S_Coil( #vjazd )
   END_RUNG
   // the same network as SCL:
   #L_zl_h := #stavL = 1;
   #L_zl_d := #L_zl_h AND NOT #smer_v1;
   #PrL_zl := #L_zl_d AND #prerusovac;
   IF #L_zl_h THEN #vjazd := TRUE; END_IF;
END_REGION

REGION Network 4: PrL
   RUNG wire#powerrail
      { S7_Templates := "SrcType := Byte" } EQ_Contact(in1 := #stavL, in2 := 0)
      wire#w1
      Coil( #PrL_zl )
   END_RUNG
   RUNG wire#powerrail
      { S7_Templates := "SrcType := Byte" } EQ_Contact(in1 := #stavL, in2 := 3)
   END_RUNG wire#w1
   RUNG wire#powerrail
      { S7_Templates := "SrcType := Byte" } EQ_Contact(in1 := #stavL, in2 := 1)
      I_Contact( #smer_v1 )
      Contact( #prerusovac )
   END_RUNG wire#w1
   RUNG wire#powerrail
      { S7_Templates := "SrcType := Byte" } EQ_Contact(in1 := #stavL, in2 := 1)
      Contact( #smer_v1 )
      Coil( #PrL_ze )
   END_RUNG
   // the same network as SCL:
   #PrL_zl := (#stavL = 0) OR (#stavL = 3) OR ((#stavL = 1) AND NOT #smer_v1 AND #prerusovac);
   #PrL_ze := (#stavL = 1) AND #smer_v1;
END_REGION

REGION Network 5: L PN
   RUNG wire#powerrail
      { S7_Templates := "SrcType := Byte" } EQ_Contact(in1 := #stavL, in2 := 3)
      Contact( #prerusovac )
      Coil( #L_bi )
   END_RUNG
   // the same network as SCL:
   #L_bi := (#stavL = 3) AND #prerusovac;
END_REGION

REGION Network 6: S1 Stoj
   RUNG wire#powerrail
      { S7_Templates := "SrcType := Byte" } EQ_Contact(in1 := #stavS1, in2 := 0)
      wire#w1
      Coil( #S1_ce )
   END_RUNG
   RUNG wire#powerrail
      { S7_Templates := "SrcType := Byte" } EQ_Contact(in1 := #stavS1, in2 := 3)
   END_RUNG wire#w1
   // the same network as SCL:
   #S1_ce := (#stavS1 = 0) OR (#stavS1 = 3);
END_REGION

REGION Network 7: S1 Volno
   RUNG wire#powerrail
      { S7_Templates := "SrcType := Byte" } EQ_Contact(in1 := #stavS1, in2 := 1)
      Coil( #S1_ze )
   END_RUNG
   // the same network as SCL:
   #S1_ze := #stavS1 = 1;
END_REGION

REGION Network 8: S1 Posun / PN
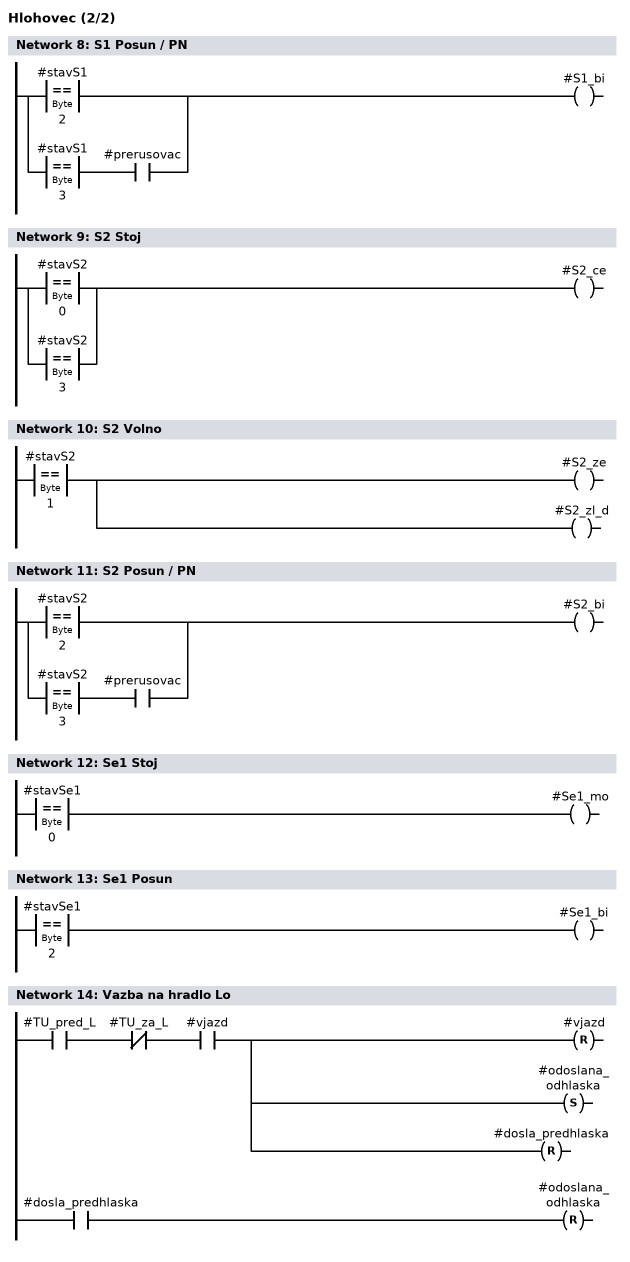
   RUNG wire#powerrail
      { S7_Templates := "SrcType := Byte" } EQ_Contact(in1 := #stavS1, in2 := 2)
      wire#w1
      Coil( #S1_bi )
   END_RUNG
   RUNG wire#powerrail
      { S7_Templates := "SrcType := Byte" } EQ_Contact(in1 := #stavS1, in2 := 3)
      Contact( #prerusovac )
   END_RUNG wire#w1
   // the same network as SCL:
   #S1_bi := (#stavS1 = 2) OR ((#stavS1 = 3) AND #prerusovac);
END_REGION

REGION Network 9: S2 Stoj
   RUNG wire#powerrail
      { S7_Templates := "SrcType := Byte" } EQ_Contact(in1 := #stavS2, in2 := 0)
      wire#w1
      Coil( #S2_ce )
   END_RUNG
   RUNG wire#powerrail
      { S7_Templates := "SrcType := Byte" } EQ_Contact(in1 := #stavS2, in2 := 3)
   END_RUNG wire#w1
   // the same network as SCL:
   #S2_ce := (#stavS2 = 0) OR (#stavS2 = 3);
END_REGION

REGION Network 10: S2 Volno
   RUNG wire#powerrail
      { S7_Templates := "SrcType := Byte" } EQ_Contact(in1 := #stavS2, in2 := 1)
      wire#w1
      Coil( #S2_ze )
   END_RUNG
   RUNG wire#w1
      Coil( #S2_zl_d )
   END_RUNG
   // the same network as SCL:
   #S2_ze := #stavS2 = 1;
   #S2_zl_d := #S2_ze;
END_REGION

REGION Network 11: S2 Posun / PN
   RUNG wire#powerrail
      { S7_Templates := "SrcType := Byte" } EQ_Contact(in1 := #stavS2, in2 := 2)
      wire#w1
      Coil( #S2_bi )
   END_RUNG
   RUNG wire#powerrail
      { S7_Templates := "SrcType := Byte" } EQ_Contact(in1 := #stavS2, in2 := 3)
      Contact( #prerusovac )
   END_RUNG wire#w1
   // the same network as SCL:
   #S2_bi := (#stavS2 = 2) OR ((#stavS2 = 3) AND #prerusovac);
END_REGION

REGION Network 12: Se1 Stoj
   RUNG wire#powerrail
      { S7_Templates := "SrcType := Byte" } EQ_Contact(in1 := #stavSe1, in2 := 0)
      Coil( #Se1_mo )
   END_RUNG
   // the same network as SCL:
   #Se1_mo := #stavSe1 = 0;
END_REGION

REGION Network 13: Se1 Posun
   RUNG wire#powerrail
      { S7_Templates := "SrcType := Byte" } EQ_Contact(in1 := #stavSe1, in2 := 2)
      Coil( #Se1_bi )
   END_RUNG
   // the same network as SCL:
   #Se1_bi := #stavSe1 = 2;
END_REGION

REGION Network 14: Vazba na hradlo Lo
   RUNG wire#powerrail
      Contact( #TU_pred_L )
      I_Contact( #TU_za_L )
      Contact( #vjazd )
      wire#w1
      R_Coil( #vjazd )
   END_RUNG
   RUNG wire#w1
      S_Coil( #odoslana_odhlaska )
   END_RUNG
   RUNG wire#w1
      R_Coil( #dosla_predhlaska )
   END_RUNG
   RUNG wire#powerrail
      Contact( #dosla_predhlaska )
      R_Coil( #odoslana_odhlaska )
   END_RUNG
   // the same network as SCL:
   #_w1 := #TU_pred_L AND NOT #TU_za_L AND #vjazd;
   IF #_w1 THEN
       #vjazd := FALSE;
       #odoslana_odhlaska := TRUE;
       #dosla_predhlaska := FALSE;
   END_IF;
   IF #dosla_predhlaska THEN #odoslana_odhlaska := FALSE; END_IF;
END_REGION
END_FUNCTION_BLOCK

FUNCTION_BLOCK "Vyhybka"   // FB7, LAD
{ S7_Optimized_Access := 'TRUE' }
VERSION : 0.1
   VAR_INPUT
      smer_Plus : Bool;   // vstup z koncoveho spinaca plus
      smer_Minus : Bool;   // vstup z koncoveho spinaca minus
   END_VAR
   VAR_OUTPUT
      prestavnik : Bool;   // ovladanie prestavnika
      smer : Bool := 1;   // data do PC
   END_VAR
   VAR_IN_OUT
      prestavenie_doM : Bool;   // prikaz z PC
      prestavenie_doP : Bool;   // prikaz z PC
      prestavenie_doP_manual : Bool;
      prestavenie_doM_manual : Bool;
   END_VAR
   VAR
      stav : Byte;
   END_VAR
BEGIN

REGION Network 1: PLUS
